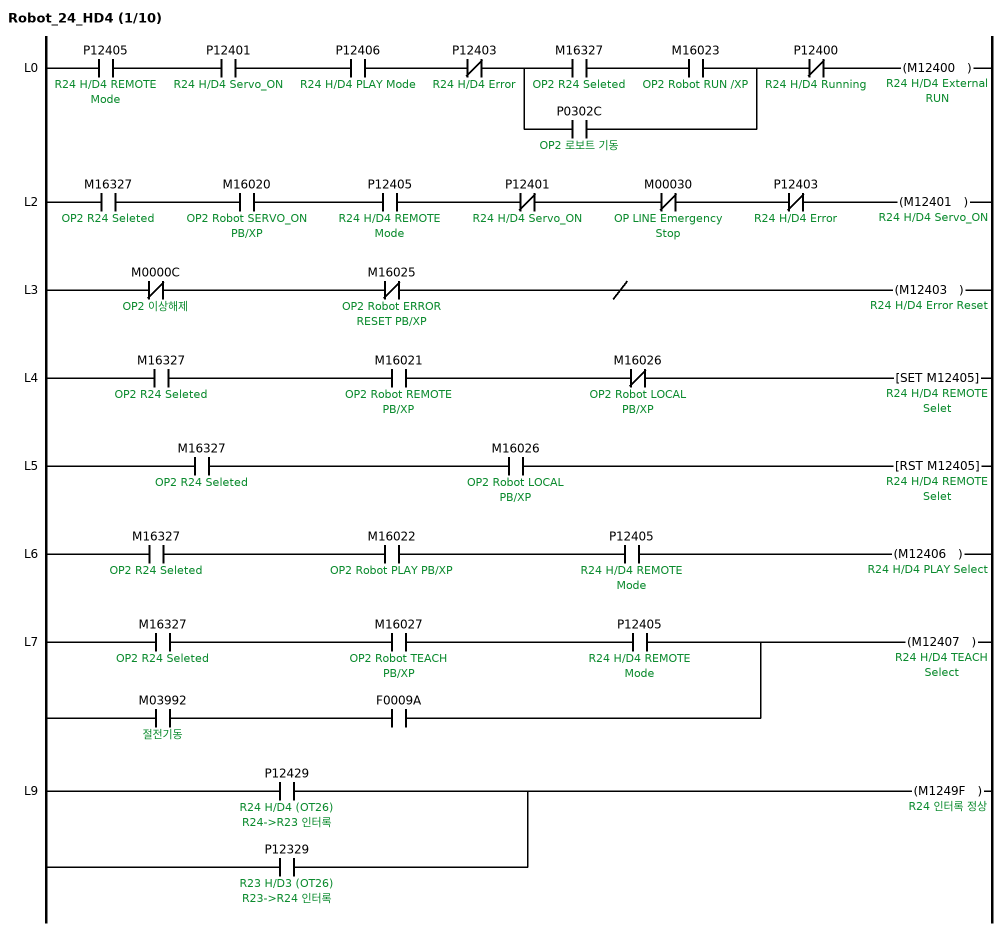
[picture p384: Robot_24_HD4 rungs L0-L9]
; L0
LOAD      P12405	// R24 H/D4 REMOTE Mode
AND       P12401	// R24 H/D4 Servo_ON
AND       P12406	// R24 H/D4 PLAY Mode
AND NOT   P12403	// R24 H/D4 Error
LOAD      M16327	// OP2 R24 Seleted
AND       M16023	// OP2 Robot RUN /XP
OR        P0302C	// OP2 로보트 기동
AND LOAD
AND NOT   P12400	// R24 H/D4 Running
OUT       M12400	// R24 H/D4 External RUN
; L2
LOAD      M16327	// OP2 R24 Seleted
AND       M16020	// OP2 Robot SERVO_ON PB/XP
AND       P12405	// R24 H/D4 REMOTE Mode
AND NOT   P12401	// R24 H/D4 Servo_ON
AND NOT   M00030	// OP LINE Emergency Stop
AND NOT   P12403	// R24 H/D4 Error
OUT       M12401	// R24 H/D4 Servo_ON
; L3
LOAD NOT  M0000C	// OP2 이상해제
AND NOT   M16025	// OP2 Robot ERROR RESET PB/XP
NOT
OUT       M12403	// R24 H/D4 Error Reset
; L4
LOAD      M16327	// OP2 R24 Seleted
AND       M16021	// OP2 Robot REMOTE PB/XP
AND NOT   M16026	// OP2 Robot LOCAL PB/XP
SET       M12405	// R24 H/D4 REMOTE Selet
; L5
LOAD      M16327	// OP2 R24 Seleted
AND       M16026	// OP2 Robot LOCAL PB/XP
RST       M12405	// R24 H/D4 REMOTE Selet
; L6
LOAD      M16327	// OP2 R24 Seleted
AND       M16022	// OP2 Robot PLAY PB/XP
AND       P12405	// R24 H/D4 REMOTE Mode
OUT       M12406	// R24 H/D4 PLAY Select
; L7
LOAD      M16327	// OP2 R24 Seleted
AND       M16027	// OP2 Robot TEACH PB/XP
AND       P12405	// R24 H/D4 REMOTE Mode
LOAD      M03992	// 절전기동
AND       F0009A
OR LOAD
OUT       M12407	// R24 H/D4 TEACH Select
; L9
LOAD      P12429	// R24 H/D4 (OT26) R24->R23 인터록
OR        P12329	// R23 H/D3 (OT26) R23->R24 인터록
OUT       M1249F	// R24 인터록 정상

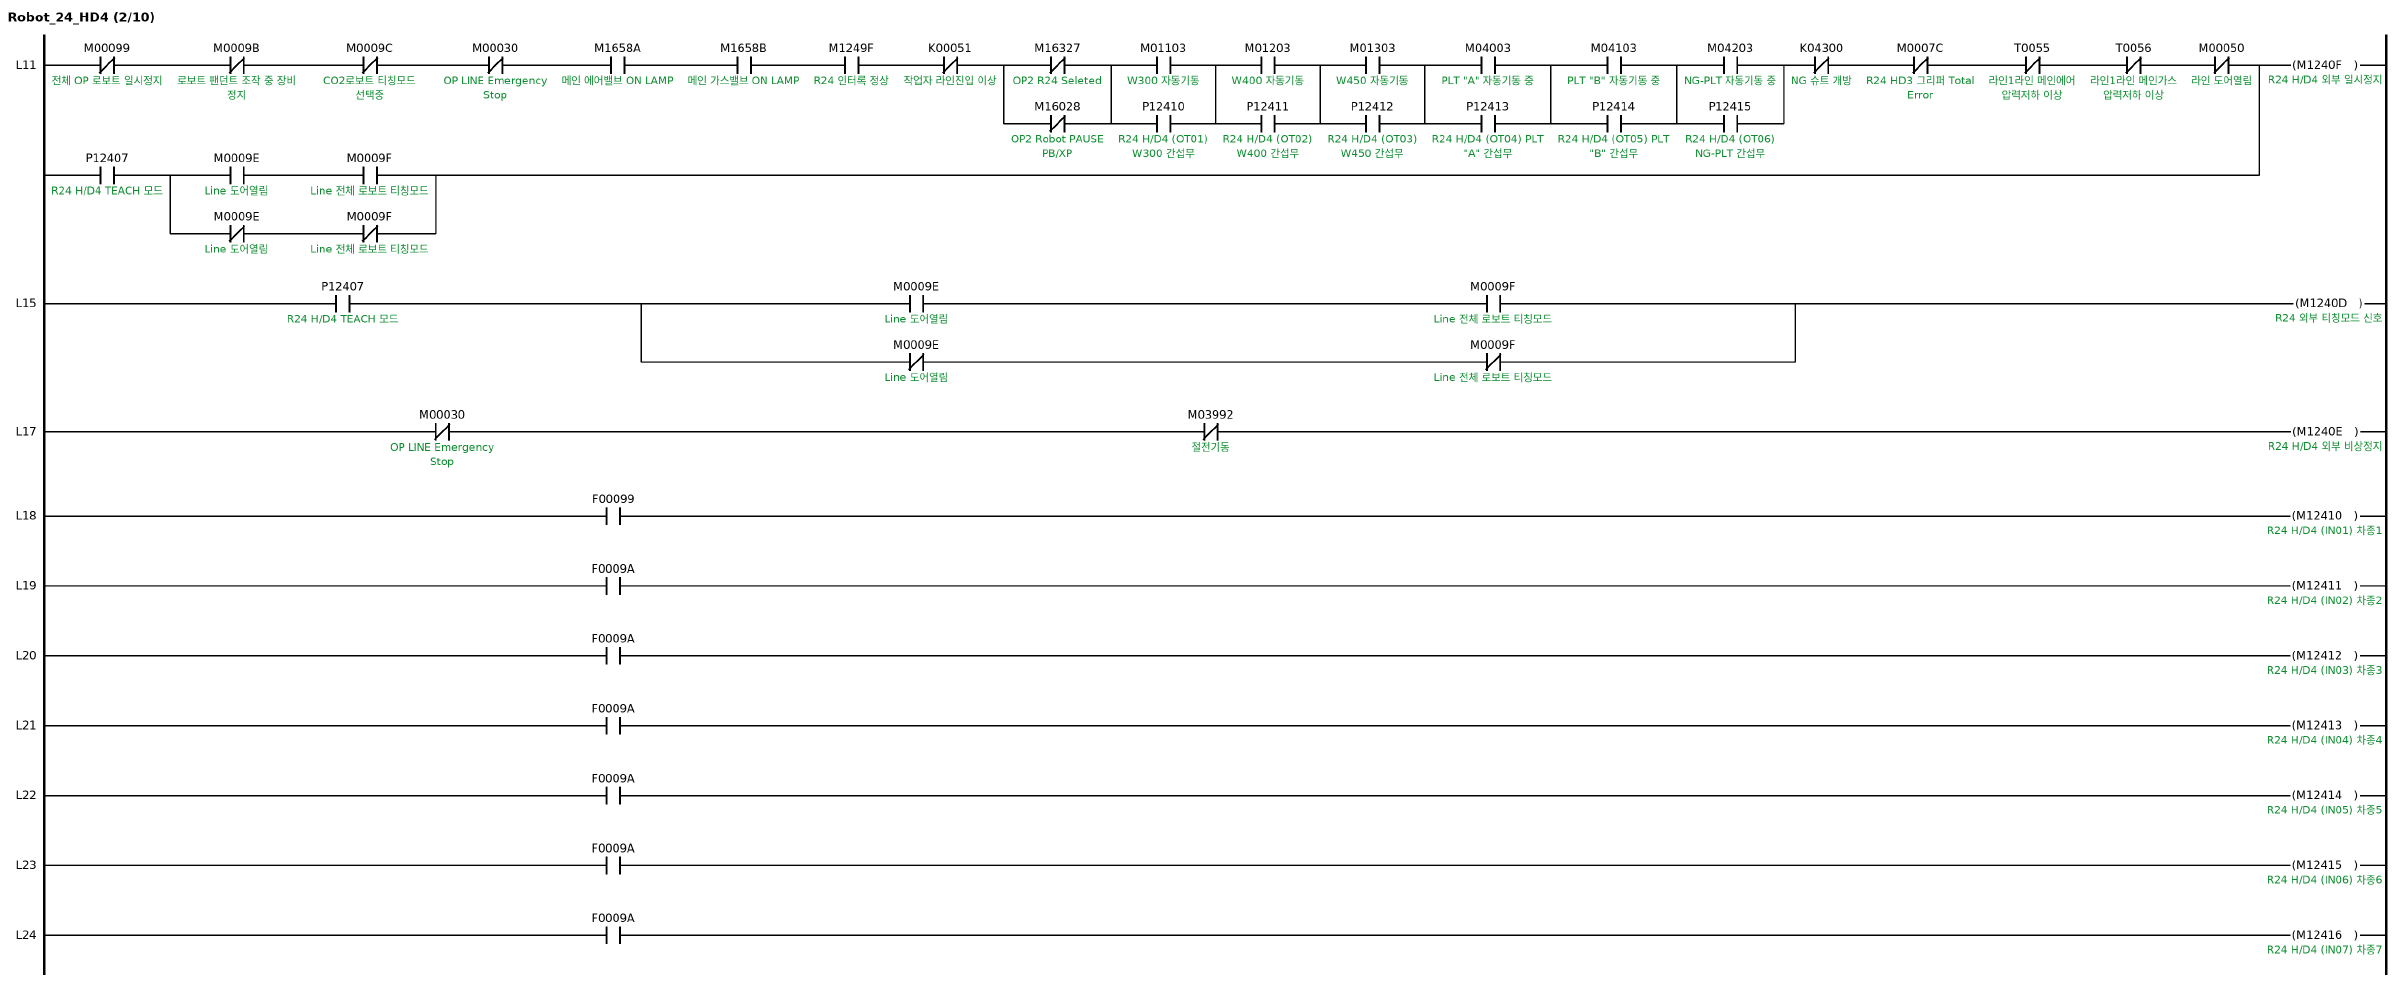
; L11
LOAD NOT  M00099	// 전체 OP 로보트 일시정지
AND NOT   M0009B	// 로보트 팬던트 조작 중 장비 정지
AND NOT   M0009C	// CO2로보트 티칭모드 선택중
AND NOT   M00030	// OP LINE Emergency Stop
AND       M1658A	// 메인 에어밸브 ON LAMP
AND       M1658B	// 메인 가스밸브 ON LAMP
AND       M1249F	// R24 인터록 정상
AND NOT   K00051	//  작업자 라인진입 이상
LOAD NOT  M16327	// OP2 R24 Seleted
OR NOT    M16028	// OP2 Robot PAUSE PB/XP
AND LOAD
LOAD      M01103	// W300 자동기동
OR        P12410	// R24 H/D4 (OT01) W300 간섭무
AND LOAD
LOAD      M01203	// W400 자동기동
OR        P12411	// R24 H/D4 (OT02) W400 간섭무
AND LOAD
LOAD      M01303	// W450 자동기동
OR        P12412	// R24 H/D4 (OT03) W450 간섭무
AND LOAD
LOAD      M04003	// PLT "A" 자동기동 중
OR        P12413	// R24 H/D4 (OT04) PLT "A" 간섭무
AND LOAD
LOAD      M04103	// PLT "B" 자동기동 중
OR        P12414	// R24 H/D4 (OT05) PLT "B" 간섭무
AND LOAD
LOAD      M04203	// NG-PLT 자동기동 중
OR        P12415	// R24 H/D4 (OT06) NG-PLT 간섭무
AND LOAD
AND NOT   K04300	// NG 슈트 개방
AND NOT   M0007C	// R24 HD3 그리퍼 Total Error 
AND NOT   T0055	// 라인1라인 메인에어 압력저하 이상
AND NOT   T0056	// 라인1라인 메인가스 압력저하 이상
AND NOT   M00050	// 라인 도어열림
LOAD      P12407	// R24 H/D4 TEACH 모드
LOAD      M0009E	// Line 도어열림
AND       M0009F	// Line 전체 로보트 티칭모드
LOAD NOT  M0009E	// Line 도어열림
AND NOT   M0009F	// Line 전체 로보트 티칭모드
OR LOAD
AND LOAD
OR LOAD
OUT       M1240F	// R24 H/D4 외부 일시정지
; L15
LOAD      P12407	// R24 H/D4 TEACH 모드
LOAD      M0009E	// Line 도어열림
AND       M0009F	// Line 전체 로보트 티칭모드
LOAD NOT  M0009E	// Line 도어열림
AND NOT   M0009F	// Line 전체 로보트 티칭모드
OR LOAD
AND LOAD
OUT       M1240D	// R24 외부 티칭모드 신호
; L17
LOAD NOT  M00030	// OP LINE Emergency Stop
AND NOT   M03992	// 절전기동
OUT       M1240E	// R24 H/D4 외부 비상정지 
; L18
LOAD      F00099
OUT       M12410	// R24 H/D4 (IN01) 차종1
; L19
LOAD      F0009A
OUT       M12411	// R24 H/D4 (IN02) 차종2
; L20
LOAD      F0009A
OUT       M12412	// R24 H/D4 (IN03) 차종3
; L21
LOAD      F0009A
OUT       M12413	// R24 H/D4 (IN04) 차종4
; L22
LOAD      F0009A
OUT       M12414	// R24 H/D4 (IN05) 차종5
; L23
LOAD      F0009A
OUT       M12415	// R24 H/D4 (IN06) 차종6
; L24
LOAD      F0009A
OUT       M12416	// R24 H/D4 (IN07) 차종7

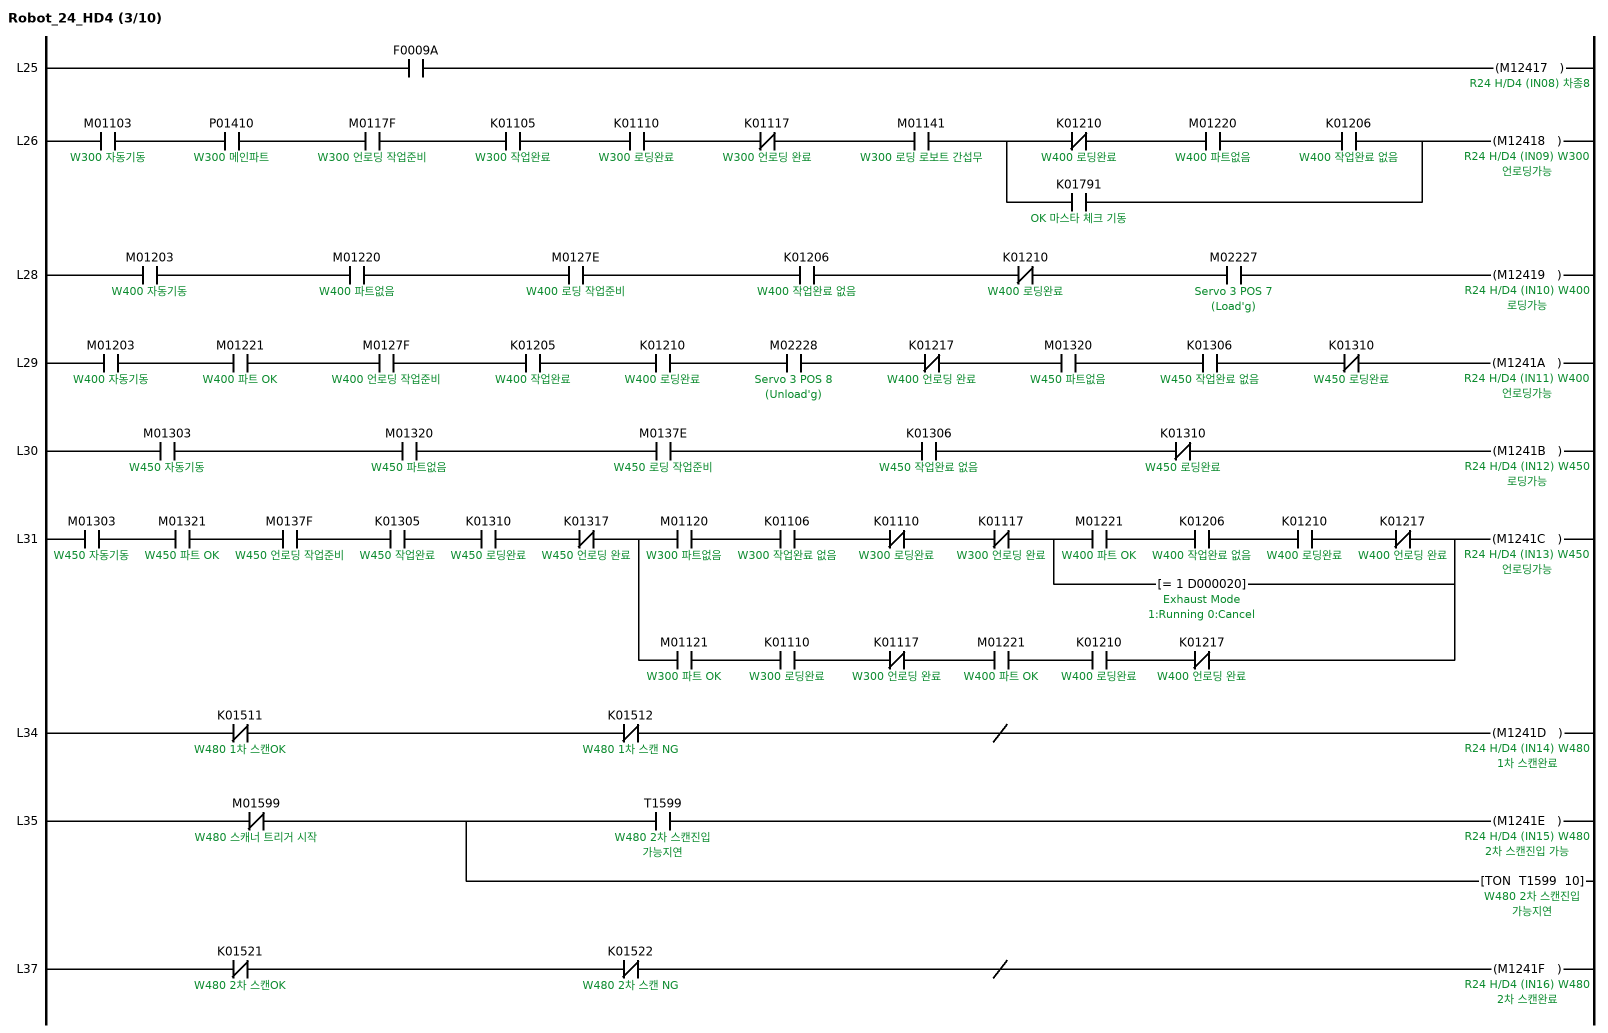
; L25
LOAD      F0009A
OUT       M12417	// R24 H/D4 (IN08) 차종8
; L26
LOAD      M01103	// W300 자동기동
AND       P01410	// W300 메인파트
AND       M0117F	// W300 언로딩 작업준비
AND       K01105	// W300 작업완료
AND       K01110	// W300 로딩완료
AND NOT   K01117	// W300 언로딩 완료
AND       M01141	// W300 로딩 로보트 간섭무
LOAD NOT  K01210	// W400 로딩완료
AND       M01220	// W400 파트없음
AND       K01206	// W400 작업완료 없음
OR        K01791	// OK 마스타 체크 기동
AND LOAD
OUT       M12418	// R24 H/D4 (IN09) W300 언로딩가능
; L28
LOAD      M01203	// W400 자동기동
AND       M01220	// W400 파트없음
AND       M0127E	// W400 로딩 작업준비
AND       K01206	// W400 작업완료 없음
AND NOT   K01210	// W400 로딩완료
AND       M02227	// Servo 3 POS 7 (Load'g)
OUT       M12419	// R24 H/D4 (IN10) W400 로딩가능
; L29
LOAD      M01203	// W400 자동기동
AND       M01221	// W400 파트 OK
AND       M0127F	// W400 언로딩 작업준비
AND       K01205	// W400 작업완료
AND       K01210	// W400 로딩완료
AND       M02228	// Servo 3 POS 8 (Unload'g)
AND NOT   K01217	// W400 언로딩 완료
AND       M01320	// W450 파트없음
AND       K01306	// W450 작업완료 없음
AND NOT   K01310	// W450 로딩완료
OUT       M1241A	// R24 H/D4 (IN11) W400 언로딩가능
; L30
LOAD      M01303	// W450 자동기동
AND       M01320	// W450 파트없음
AND       M0137E	// W450 로딩 작업준비
AND       K01306	// W450 작업완료 없음
AND NOT   K01310	// W450 로딩완료
OUT       M1241B	// R24 H/D4 (IN12) W450 로딩가능
; L31
LOAD      M01303	// W450 자동기동
AND       M01321	// W450 파트 OK
AND       M0137F	// W450 언로딩 작업준비
AND       K01305	// W450 작업완료
AND       K01310	// W450 로딩완료
AND NOT   K01317	// W450 언로딩 완료
LOAD      M01120	// W300 파트없음
AND       K01106	// W300 작업완료 없음
AND NOT   K01110	// W300 로딩완료
AND NOT   K01117	// W300 언로딩 완료
LOAD      M01221	// W400 파트 OK
AND       K01206	// W400 작업완료 없음
AND       K01210	// W400 로딩완료
AND NOT   K01217	// W400 언로딩 완료
OR=       1 D000020	// Exhaust Mode 1:Running 0:Cancel
AND LOAD
LOAD      M01121	// W300 파트 OK
AND       K01110	// W300 로딩완료
AND NOT   K01117	// W300 언로딩 완료
AND       M01221	// W400 파트 OK
AND       K01210	// W400 로딩완료
AND NOT   K01217	// W400 언로딩 완료
OR LOAD
AND LOAD
OUT       M1241C	// R24 H/D4 (IN13) W450 언로딩가능
; L34
LOAD NOT  K01511	// W480 1차 스캔OK
AND NOT   K01512	// W480 1차 스캔 NG
NOT
OUT       M1241D	// R24 H/D4 (IN14) W480 1차 스캔완료
; L35
LOAD NOT  M01599	// W480 스캐너 트리거 시작
MPUSH
AND       T1599	// W480 2차 스캔진입 가능지연
OUT       M1241E	// R24 H/D4 (IN15) W480 2차 스캔진입 가능
MPOP
TON       T1599 10	// W480 2차 스캔진입 가능지연
; L37
LOAD NOT  K01521	// W480 2차 스캔OK
AND NOT   K01522	// W480 2차 스캔 NG
NOT
OUT       M1241F	// R24 H/D4 (IN16) W480 2차 스캔완료

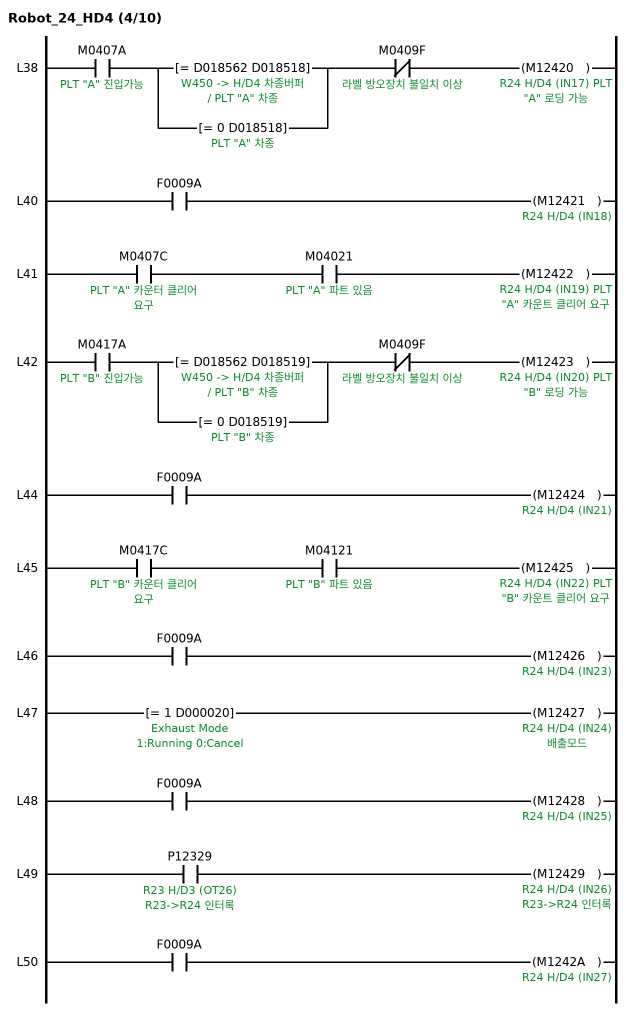
; L38
LOAD      M0407A	// PLT "A" 진입가능
LOAD=     D018562 D018518	// W450 -> H/D4 차종버퍼 / PLT "A" 차종
OR=       0 D018518	// PLT "A" 차종
AND LOAD
AND NOT   M0409F	// 라벨 방오장치 불일치 이상
OUT       M12420	// R24 H/D4 (IN17) PLT "A" 로딩 가능
; L40
LOAD      F0009A
OUT       M12421	// R24 H/D4 (IN18)
; L41
LOAD      M0407C	// PLT "A" 카운터 클리어 요구
AND       M04021	// PLT "A" 파트 있음
OUT       M12422	// R24 H/D4 (IN19) PLT "A" 카운트 클리어 요구
; L42
LOAD      M0417A	// PLT "B" 진입가능
LOAD=     D018562 D018519	// W450 -> H/D4 차종버퍼 / PLT "B" 차종
OR=       0 D018519	// PLT "B" 차종
AND LOAD
AND NOT   M0409F	// 라벨 방오장치 불일치 이상
OUT       M12423	// R24 H/D4 (IN20) PLT "B" 로딩 가능
; L44
LOAD      F0009A
OUT       M12424	// R24 H/D4 (IN21)
; L45
LOAD      M0417C	// PLT "B" 카운터 클리어 요구
AND       M04121	// PLT "B" 파트 있음
OUT       M12425	// R24 H/D4 (IN22) PLT "B" 카운트 클리어 요구
; L46
LOAD      F0009A
OUT       M12426	// R24 H/D4 (IN23)
; L47
LOAD=     1 D000020	// Exhaust Mode 1:Running 0:Cancel
OUT       M12427	// R24 H/D4 (IN24) 배출모드
; L48
LOAD      F0009A
OUT       M12428	// R24 H/D4 (IN25)
; L49
LOAD      P12329	// R23 H/D3 (OT26) R23->R24 인터록
OUT       M12429	// R24 H/D4 (IN26) R23->R24 인터록
; L50
LOAD      F0009A
OUT       M1242A	// R24 H/D4 (IN27)

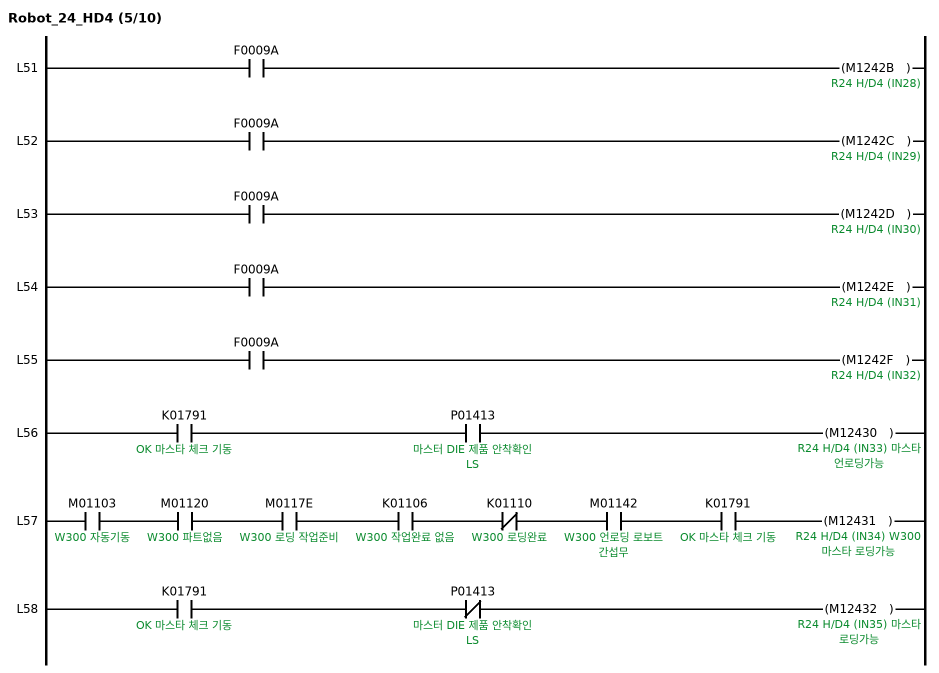
; L51
LOAD      F0009A
OUT       M1242B	// R24 H/D4 (IN28)
; L52
LOAD      F0009A
OUT       M1242C	// R24 H/D4 (IN29)
; L53
LOAD      F0009A
OUT       M1242D	// R24 H/D4 (IN30)
; L54
LOAD      F0009A
OUT       M1242E	// R24 H/D4 (IN31)
; L55
LOAD      F0009A
OUT       M1242F	// R24 H/D4 (IN32)
; L56
LOAD      K01791	// OK 마스타 체크 기동
AND       P01413	// 마스터 DIE 제품 안착확인 LS
OUT       M12430	// R24 H/D4 (IN33) 마스타 언로딩가능
; L57
LOAD      M01103	// W300 자동기동
AND       M01120	// W300 파트없음
AND       M0117E	// W300 로딩 작업준비
AND       K01106	// W300 작업완료 없음
AND NOT   K01110	// W300 로딩완료
AND       M01142	// W300 언로딩 로보트 간섭무
AND       K01791	// OK 마스타 체크 기동
OUT       M12431	// R24 H/D4 (IN34) W300 마스타 로딩가능
; L58
LOAD      K01791	// OK 마스타 체크 기동
AND NOT   P01413	// 마스터 DIE 제품 안착확인 LS
OUT       M12432	// R24 H/D4 (IN35) 마스타 로딩가능

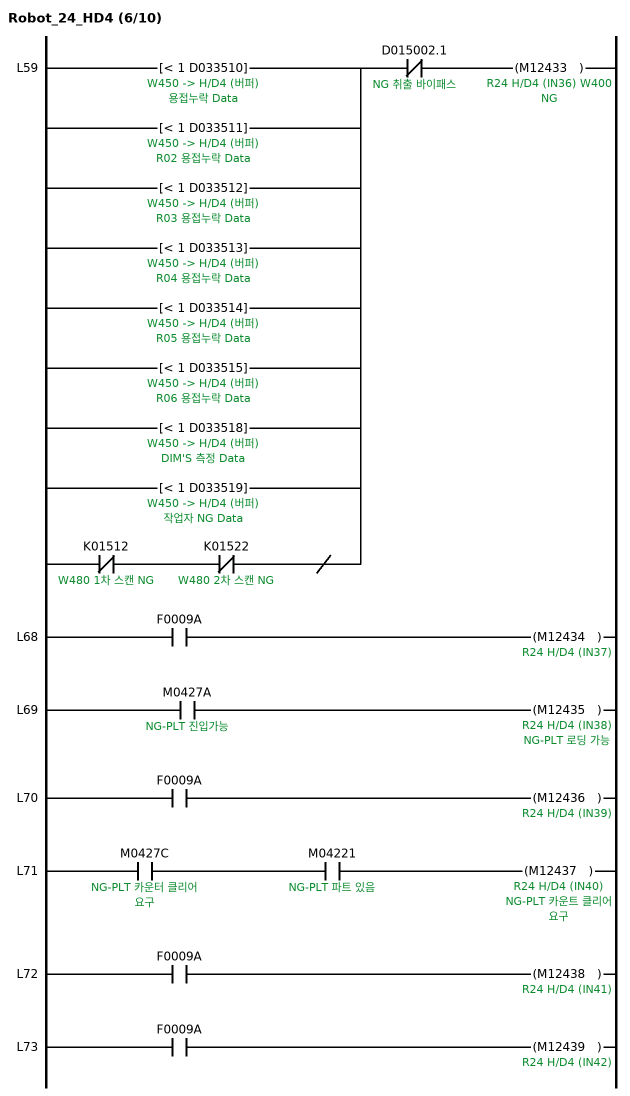
; L59
LOAD<     1 D033510	// W450 -> H/D4 (버퍼) 용접누락 Data
OR<       1 D033511	// W450 -> H/D4 (버퍼) R02 용접누락 Data
OR<       1 D033512	// W450 -> H/D4 (버퍼) R03 용접누락 Data
OR<       1 D033513	// W450 -> H/D4 (버퍼) R04 용접누락 Data
OR<       1 D033514	// W450 -> H/D4 (버퍼) R05 용접누락 Data
OR<       1 D033515	// W450 -> H/D4 (버퍼) R06 용접누락 Data
OR<       1 D033518	// W450 -> H/D4 (버퍼) DIM'S 측정 Data
OR<       1 D033519	// W450 -> H/D4 (버퍼) 작업자 NG Data
LOAD NOT  K01512	// W480 1차 스캔 NG
AND NOT   K01522	// W480 2차 스캔 NG
NOT
OR LOAD
AND NOT   D015002.1	// NG 취출 바이패스
OUT       M12433	// R24 H/D4 (IN36) W400 NG
; L68
LOAD      F0009A
OUT       M12434	// R24 H/D4 (IN37)
; L69
LOAD      M0427A	// NG-PLT 진입가능
OUT       M12435	// R24 H/D4 (IN38) NG-PLT 로딩 가능
; L70
LOAD      F0009A
OUT       M12436	// R24 H/D4 (IN39)
; L71
LOAD      M0427C	// NG-PLT 카운터 클리어 요구
AND       M04221	// NG-PLT 파트 있음
OUT       M12437	// R24 H/D4 (IN40) NG-PLT 카운트 클리어 요구
; L72
LOAD      F0009A
OUT       M12438	// R24 H/D4 (IN41)
; L73
LOAD      F0009A
OUT       M12439	// R24 H/D4 (IN42)

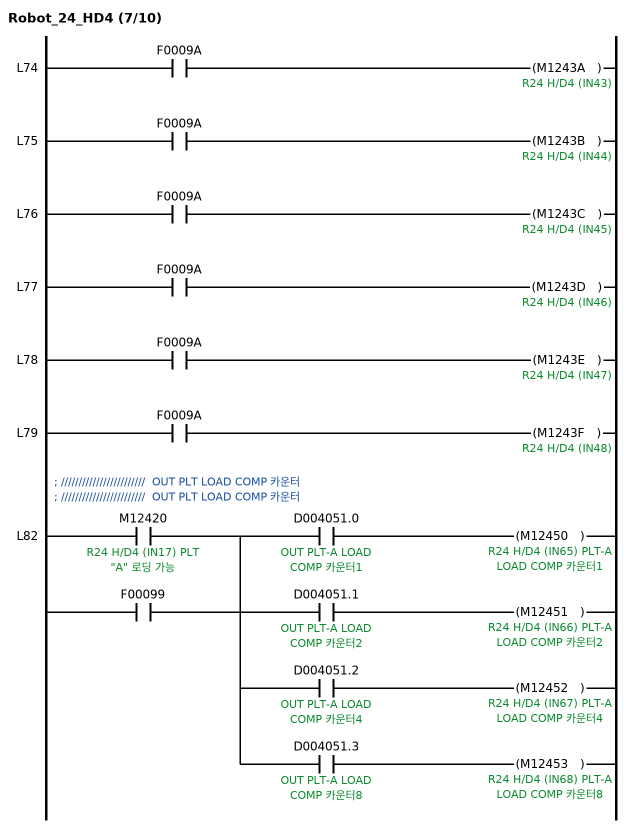
; L74
LOAD      F0009A
OUT       M1243A	// R24 H/D4 (IN43)
; L75
LOAD      F0009A
OUT       M1243B	// R24 H/D4 (IN44)
; L76
LOAD      F0009A
OUT       M1243C	// R24 H/D4 (IN45)
; L77
LOAD      F0009A
OUT       M1243D	// R24 H/D4 (IN46)
; L78
LOAD      F0009A
OUT       M1243E	// R24 H/D4 (IN47)
; L79
LOAD      F0009A
OUT       M1243F	// R24 H/D4 (IN48)
// ////////////////////////  OUT PLT LOAD COMP 카운터
// ////////////////////////  OUT PLT LOAD COMP 카운터
; L82
LOAD      M12420	// R24 H/D4 (IN17) PLT "A" 로딩 가능
OR        F00099
MPUSH
AND       D004051.0	// OUT PLT-A LOAD COMP 카운터1
OUT       M12450	// R24 H/D4 (IN65) PLT-A LOAD COMP 카운터1
MLOAD
AND       D004051.1	// OUT PLT-A LOAD COMP 카운터2
OUT       M12451	// R24 H/D4 (IN66) PLT-A LOAD COMP 카운터2
MLOAD
AND       D004051.2	// OUT PLT-A LOAD COMP 카운터4
OUT       M12452	// R24 H/D4 (IN67) PLT-A LOAD COMP 카운터4
MPOP
AND       D004051.3	// OUT PLT-A LOAD COMP 카운터8
OUT       M12453	// R24 H/D4 (IN68) PLT-A LOAD COMP 카운터8

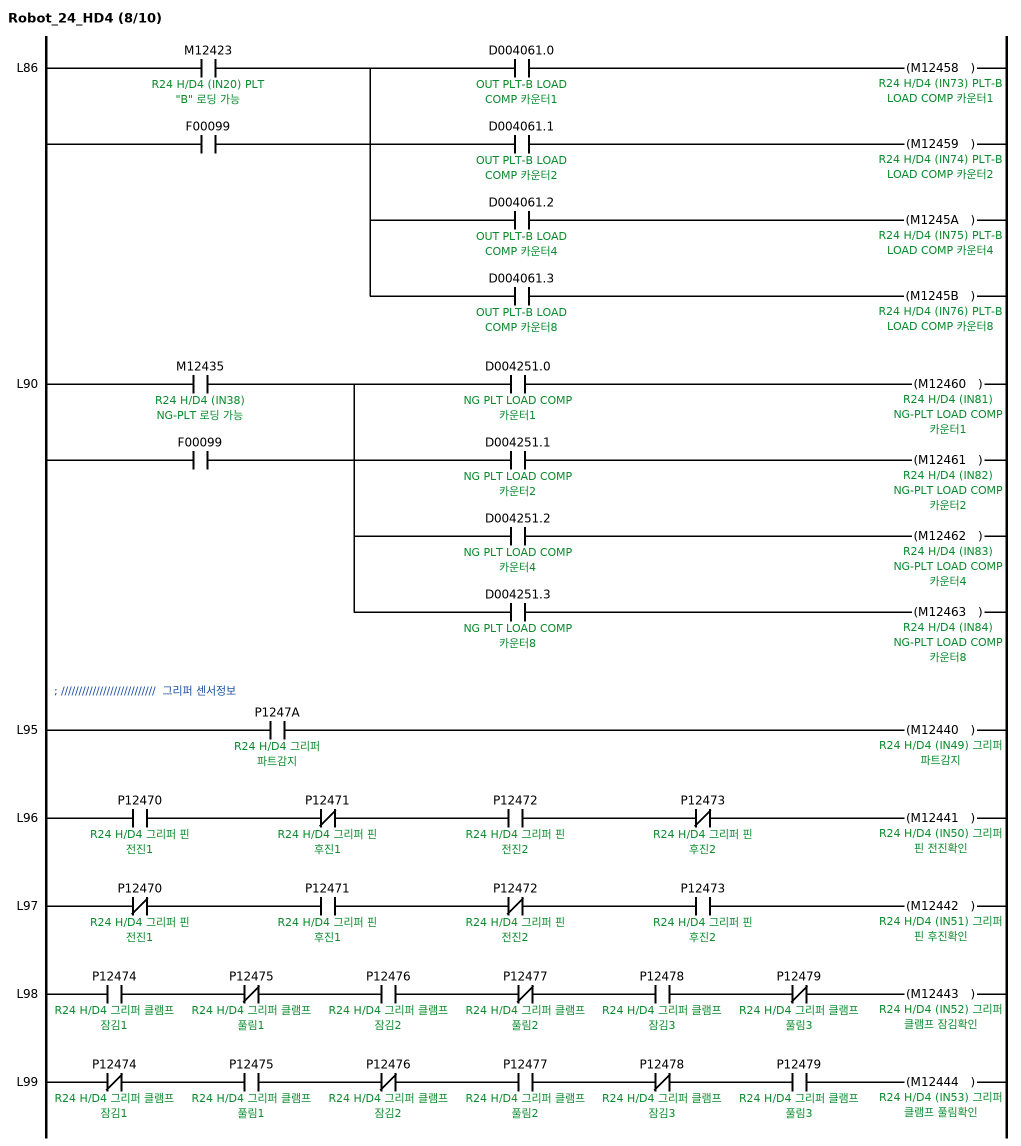
; L86
LOAD      M12423	// R24 H/D4 (IN20) PLT "B" 로딩 가능
OR        F00099
MPUSH
AND       D004061.0	// OUT PLT-B LOAD COMP 카운터1
OUT       M12458	// R24 H/D4 (IN73) PLT-B LOAD COMP 카운터1
MLOAD
AND       D004061.1	// OUT PLT-B LOAD COMP 카운터2
OUT       M12459	// R24 H/D4 (IN74) PLT-B LOAD COMP 카운터2
MLOAD
AND       D004061.2	// OUT PLT-B LOAD COMP 카운터4
OUT       M1245A	// R24 H/D4 (IN75) PLT-B LOAD COMP 카운터4
MPOP
AND       D004061.3	// OUT PLT-B LOAD COMP 카운터8
OUT       M1245B	// R24 H/D4 (IN76) PLT-B LOAD COMP 카운터8
; L90
LOAD      M12435	// R24 H/D4 (IN38) NG-PLT 로딩 가능
OR        F00099
MPUSH
AND       D004251.0	// NG PLT LOAD COMP 카운터1
OUT       M12460	// R24 H/D4 (IN81) NG-PLT LOAD COMP 카운터1
MLOAD
AND       D004251.1	// NG PLT LOAD COMP 카운터2
OUT       M12461	// R24 H/D4 (IN82) NG-PLT LOAD COMP 카운터2
MLOAD
AND       D004251.2	// NG PLT LOAD COMP 카운터4
OUT       M12462	// R24 H/D4 (IN83) NG-PLT LOAD COMP 카운터4
MPOP
AND       D004251.3	// NG PLT LOAD COMP 카운터8
OUT       M12463	// R24 H/D4 (IN84) NG-PLT LOAD COMP 카운터8
// ///////////////////////////  그리퍼 센서정보
; L95
LOAD      P1247A	// R24 H/D4 그리퍼 파트감지
OUT       M12440	// R24 H/D4 (IN49) 그리퍼 파트감지
; L96
LOAD      P12470	// R24 H/D4 그리퍼 핀 전진1
AND NOT   P12471	// R24 H/D4 그리퍼 핀 후진1
AND       P12472	// R24 H/D4 그리퍼 핀 전진2
AND NOT   P12473	// R24 H/D4 그리퍼 핀 후진2
OUT       M12441	// R24 H/D4 (IN50) 그리퍼 핀 전진확인
; L97
LOAD NOT  P12470	// R24 H/D4 그리퍼 핀 전진1
AND       P12471	// R24 H/D4 그리퍼 핀 후진1
AND NOT   P12472	// R24 H/D4 그리퍼 핀 전진2
AND       P12473	// R24 H/D4 그리퍼 핀 후진2
OUT       M12442	// R24 H/D4 (IN51) 그리퍼 핀 후진확인
; L98
LOAD      P12474	// R24 H/D4 그리퍼 클램프 잠김1
AND NOT   P12475	// R24 H/D4 그리퍼 클램프 풀림1
AND       P12476	// R24 H/D4 그리퍼 클램프 잠김2
AND NOT   P12477	// R24 H/D4 그리퍼 클램프 풀림2
AND       P12478	// R24 H/D4 그리퍼 클램프 잠김3
AND NOT   P12479	// R24 H/D4 그리퍼 클램프 풀림3
OUT       M12443	// R24 H/D4 (IN52) 그리퍼 클램프 잠김확인
; L99
LOAD NOT  P12474	// R24 H/D4 그리퍼 클램프 잠김1
AND       P12475	// R24 H/D4 그리퍼 클램프 풀림1
AND NOT   P12476	// R24 H/D4 그리퍼 클램프 잠김2
AND       P12477	// R24 H/D4 그리퍼 클램프 풀림2
AND NOT   P12478	// R24 H/D4 그리퍼 클램프 잠김3
AND       P12479	// R24 H/D4 그리퍼 클램프 풀림3
OUT       M12444	// R24 H/D4 (IN53) 그리퍼 클램프 풀림확인

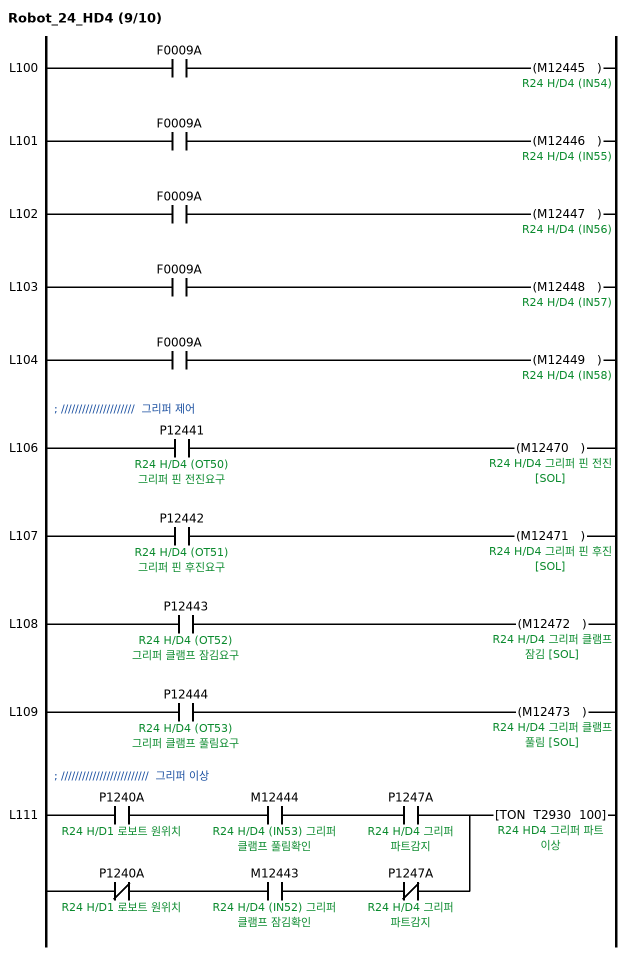
; L100
LOAD      F0009A
OUT       M12445	// R24 H/D4 (IN54)
; L101
LOAD      F0009A
OUT       M12446	// R24 H/D4 (IN55)
; L102
LOAD      F0009A
OUT       M12447	// R24 H/D4 (IN56)
; L103
LOAD      F0009A
OUT       M12448	// R24 H/D4 (IN57)
; L104
LOAD      F0009A
OUT       M12449	// R24 H/D4 (IN58)
// /////////////////////  그리퍼 제어
; L106
LOAD      P12441	// R24 H/D4 (OT50) 그리퍼 핀 전진요구
OUT       M12470	// R24 H/D4 그리퍼 핀 전진 [SOL]
; L107
LOAD      P12442	// R24 H/D4 (OT51) 그리퍼 핀 후진요구
OUT       M12471	// R24 H/D4 그리퍼 핀 후진 [SOL]
; L108
LOAD      P12443	// R24 H/D4 (OT52) 그리퍼 클램프 잠김요구
OUT       M12472	// R24 H/D4 그리퍼 클램프 잠김 [SOL]
; L109
LOAD      P12444	// R24 H/D4 (OT53) 그리퍼 클램프 풀림요구
OUT       M12473	// R24 H/D4 그리퍼 클램프 풀림 [SOL]
// /////////////////////////  그리퍼 이상
; L111
LOAD      P1240A	// R24 H/D1 로보트 원위치
AND       M12444	// R24 H/D4 (IN53) 그리퍼 클램프 풀림확인
AND       P1247A	// R24 H/D4 그리퍼 파트감지
LOAD NOT  P1240A	// R24 H/D1 로보트 원위치
AND       M12443	// R24 H/D4 (IN52) 그리퍼 클램프 잠김확인
AND NOT   P1247A	// R24 H/D4 그리퍼 파트감지
OR LOAD
TON       T2930 100	// R24 HD4 그리퍼 파트 이상

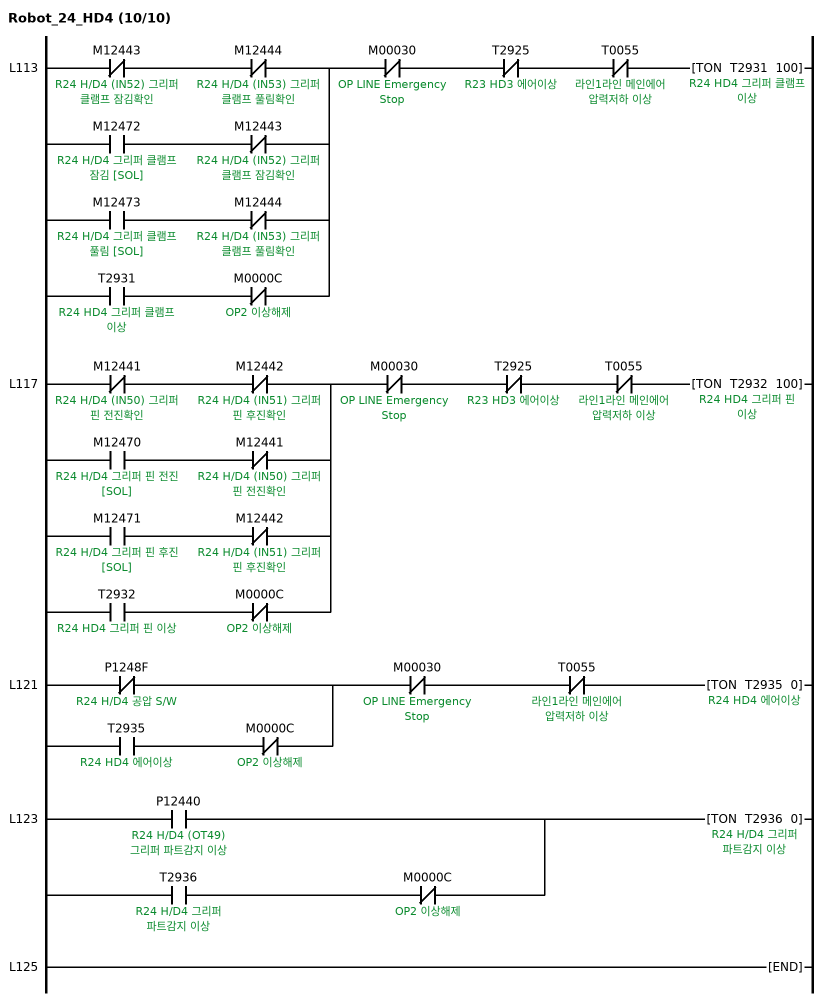
; L113
LOAD NOT  M12443	// R24 H/D4 (IN52) 그리퍼 클램프 잠김확인
AND NOT   M12444	// R24 H/D4 (IN53) 그리퍼 클램프 풀림확인
LOAD      M12472	// R24 H/D4 그리퍼 클램프 잠김 [SOL]
AND NOT   M12443	// R24 H/D4 (IN52) 그리퍼 클램프 잠김확인
OR LOAD
LOAD      M12473	// R24 H/D4 그리퍼 클램프 풀림 [SOL]
AND NOT   M12444	// R24 H/D4 (IN53) 그리퍼 클램프 풀림확인
OR LOAD
LOAD      T2931	// R24 HD4 그리퍼 클램프 이상
AND NOT   M0000C	// OP2 이상해제
OR LOAD
AND NOT   M00030	// OP LINE Emergency Stop
AND NOT   T2925	// R23 HD3 에어이상
AND NOT   T0055	// 라인1라인 메인에어 압력저하 이상
TON       T2931 100	// R24 HD4 그리퍼 클램프 이상
; L117
LOAD NOT  M12441	// R24 H/D4 (IN50) 그리퍼 핀 전진확인
AND NOT   M12442	// R24 H/D4 (IN51) 그리퍼 핀 후진확인
LOAD      M12470	// R24 H/D4 그리퍼 핀 전진 [SOL]
AND NOT   M12441	// R24 H/D4 (IN50) 그리퍼 핀 전진확인
OR LOAD
LOAD      M12471	// R24 H/D4 그리퍼 핀 후진 [SOL]
AND NOT   M12442	// R24 H/D4 (IN51) 그리퍼 핀 후진확인
OR LOAD
LOAD      T2932	// R24 HD4 그리퍼 핀 이상
AND NOT   M0000C	// OP2 이상해제
OR LOAD
AND NOT   M00030	// OP LINE Emergency Stop
AND NOT   T2925	// R23 HD3 에어이상
AND NOT   T0055	// 라인1라인 메인에어 압력저하 이상
TON       T2932 100	// R24 HD4 그리퍼 핀 이상
; L121
LOAD NOT  P1248F	// R24 H/D4 공압 S/W
LOAD      T2935	// R24 HD4 에어이상
AND NOT   M0000C	// OP2 이상해제
OR LOAD
AND NOT   M00030	// OP LINE Emergency Stop
AND NOT   T0055	// 라인1라인 메인에어 압력저하 이상
TON       T2935 0	// R24 HD4 에어이상
; L123
LOAD      P12440	// R24 H/D4 (OT49) 그리퍼 파트감지 이상
LOAD      T2936	// R24 H/D4 그리퍼 파트감지 이상
AND NOT   M0000C	// OP2 이상해제
OR LOAD
TON       T2936 0	// R24 H/D4 그리퍼 파트감지 이상
; L125
END

PROGRAM ARC관리 (task: 스캔 프로그램)

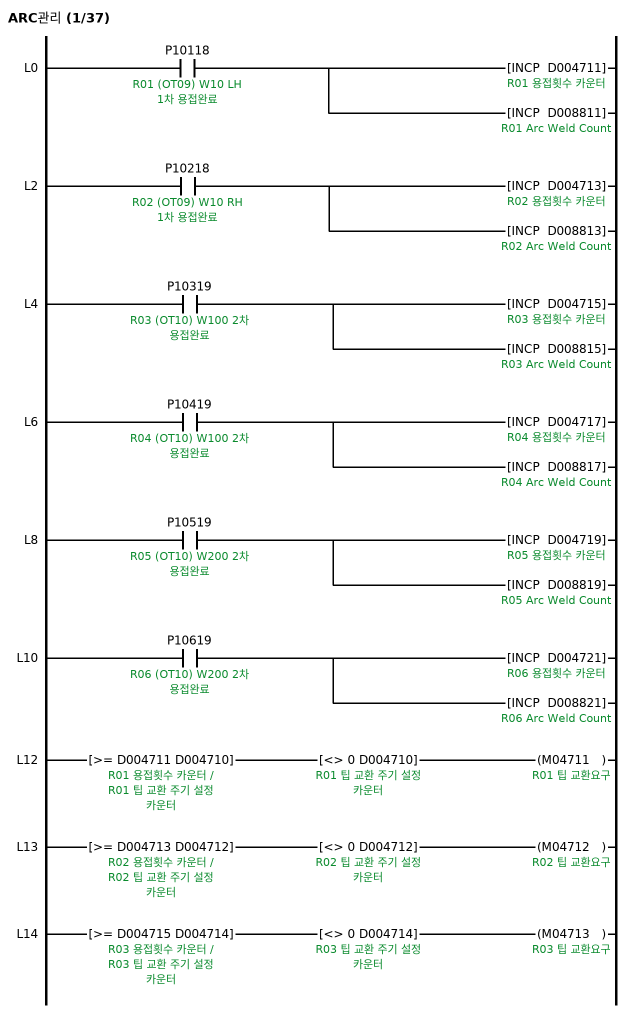
; L0
LOAD      P10118	// R01 (OT09) W10 LH 1차 용접완료
INCP      D004711	// R01 용접횟수 카운터
INCP      D008811	// R01 Arc Weld Count
; L2
LOAD      P10218	// R02 (OT09) W10 RH 1차 용접완료
INCP      D004713	// R02 용접횟수 카운터
INCP      D008813	// R02 Arc Weld Count
; L4
LOAD      P10319	// R03 (OT10) W100 2차 용접완료
INCP      D004715	// R03 용접횟수 카운터
INCP      D008815	// R03 Arc Weld Count
; L6
LOAD      P10419	// R04 (OT10) W100 2차 용접완료
INCP      D004717	// R04 용접횟수 카운터
INCP      D008817	// R04 Arc Weld Count
; L8
LOAD      P10519	// R05 (OT10) W200 2차 용접완료
INCP      D004719	// R05 용접횟수 카운터
INCP      D008819	// R05 Arc Weld Count
; L10
LOAD      P10619	// R06 (OT10) W200 2차 용접완료
INCP      D004721	// R06 용접횟수 카운터
INCP      D008821	// R06 Arc Weld Count
; L12
LOAD>=    D004711 D004710	// R01 용접횟수 카운터 / R01 팁 교환 주기 설정 카운터
AND<>     0 D004710	// R01 팁 교환 주기 설정 카운터
OUT       M04711	// R01 팁 교환요구
; L13
LOAD>=    D004713 D004712	// R02 용접횟수 카운터 / R02 팁 교환 주기 설정 카운터
AND<>     0 D004712	// R02 팁 교환 주기 설정 카운터
OUT       M04712	// R02 팁 교환요구
; L14
LOAD>=    D004715 D004714	// R03 용접횟수 카운터 / R03 팁 교환 주기 설정 카운터
AND<>     0 D004714	// R03 팁 교환 주기 설정 카운터
OUT       M04713	// R03 팁 교환요구

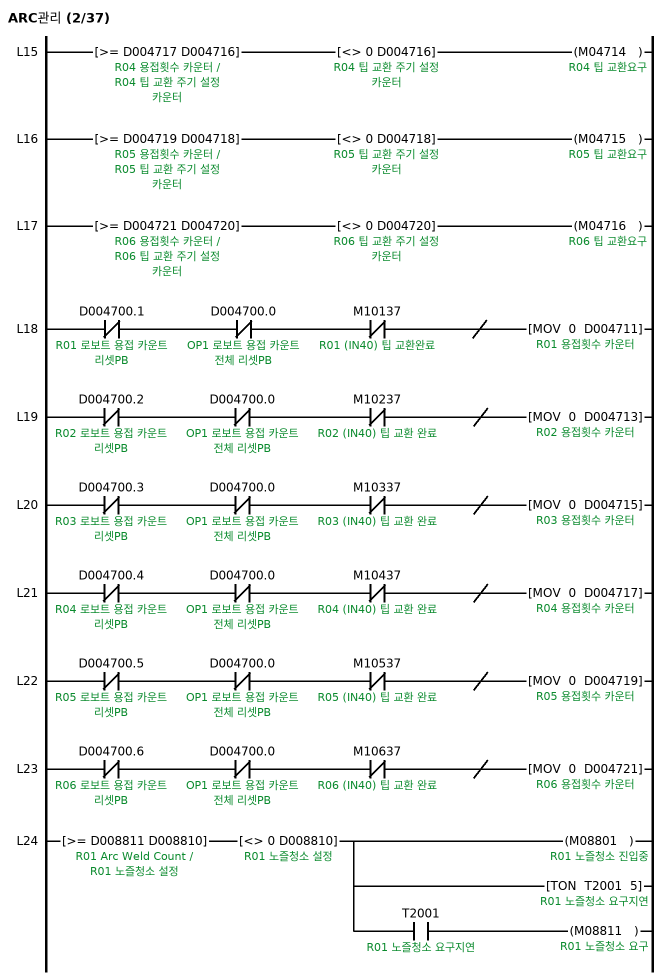
; L15
LOAD>=    D004717 D004716	// R04 용접횟수 카운터 / R04 팁 교환 주기 설정 카운터
AND<>     0 D004716	// R04 팁 교환 주기 설정 카운터
OUT       M04714	// R04 팁 교환요구
; L16
LOAD>=    D004719 D004718	// R05 용접횟수 카운터 / R05 팁 교환 주기 설정 카운터
AND<>     0 D004718	// R05 팁 교환 주기 설정 카운터
OUT       M04715	// R05 팁 교환요구
; L17
LOAD>=    D004721 D004720	// R06 용접횟수 카운터 / R06 팁 교환 주기 설정 카운터
AND<>     0 D004720	// R06 팁 교환 주기 설정 카운터
OUT       M04716	// R06 팁 교환요구
; L18
LOAD NOT  D004700.1	// R01 로보트 용접 카운트 리셋PB
AND NOT   D004700.0	// OP1 로보트 용접 카운트 전체 리셋PB
AND NOT   M10137	// R01 (IN40) 팁 교환완료
NOT
MOV       0 D004711	// R01 용접횟수 카운터
; L19
LOAD NOT  D004700.2	// R02 로보트 용접 카운트 리셋PB
AND NOT   D004700.0	// OP1 로보트 용접 카운트 전체 리셋PB
AND NOT   M10237	// R02 (IN40) 팁 교환 완료
NOT
MOV       0 D004713	// R02 용접횟수 카운터
; L20
LOAD NOT  D004700.3	// R03 로보트 용접 카운트 리셋PB
AND NOT   D004700.0	// OP1 로보트 용접 카운트 전체 리셋PB
AND NOT   M10337	// R03 (IN40) 팁 교환 완료
NOT
MOV       0 D004715	// R03 용접횟수 카운터
; L21
LOAD NOT  D004700.4	// R04 로보트 용접 카운트 리셋PB
AND NOT   D004700.0	// OP1 로보트 용접 카운트 전체 리셋PB
AND NOT   M10437	// R04 (IN40) 팁 교환 완료
NOT
MOV       0 D004717	// R04 용접횟수 카운터
; L22
LOAD NOT  D004700.5	// R05 로보트 용접 카운트 리셋PB
AND NOT   D004700.0	// OP1 로보트 용접 카운트 전체 리셋PB
AND NOT   M10537	// R05 (IN40) 팁 교환 완료
NOT
MOV       0 D004719	// R05 용접횟수 카운터
; L23
LOAD NOT  D004700.6	// R06 로보트 용접 카운트 리셋PB
AND NOT   D004700.0	// OP1 로보트 용접 카운트 전체 리셋PB
AND NOT   M10637	// R06 (IN40) 팁 교환 완료
NOT
MOV       0 D004721	// R06 용접횟수 카운터
; L24
LOAD>=    D008811 D008810	// R01 Arc Weld Count / R01 노즐청소 설정
AND<>     0 D008810	// R01 노즐청소 설정
OUT       M08801	// R01 노즐청소 진입중
TON       T2001 5	// R01 노즐청소 요구지연
AND       T2001	// R01 노즐청소 요구지연
OUT       M08811	// R01 노즐청소 요구

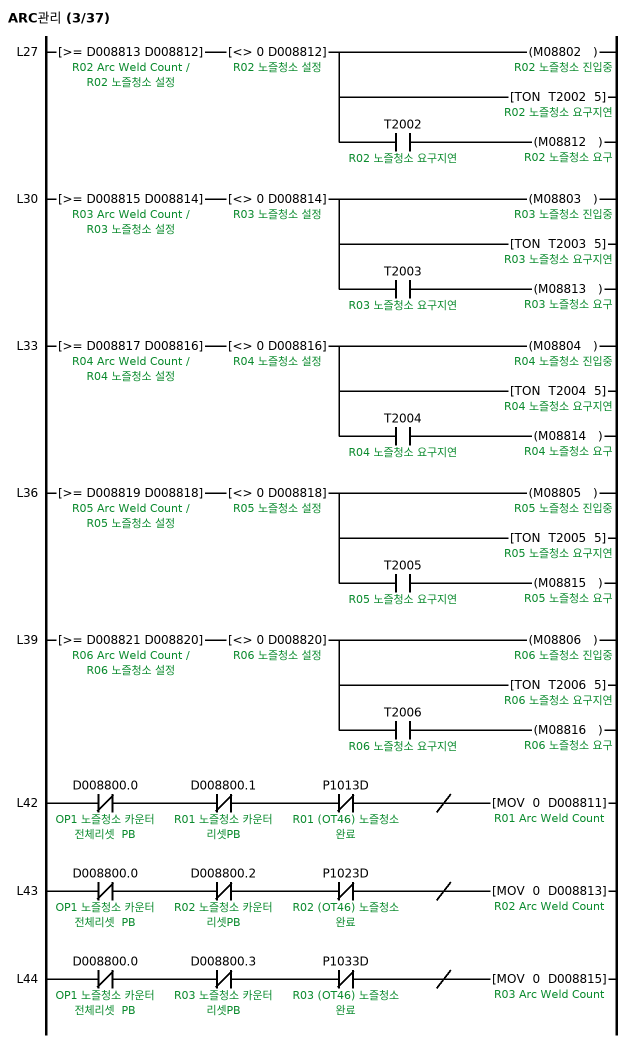
; L27
LOAD>=    D008813 D008812	// R02 Arc Weld Count / R02 노즐청소 설정
AND<>     0 D008812	// R02 노즐청소 설정
OUT       M08802	// R02 노즐청소 진입중
TON       T2002 5	// R02 노즐청소 요구지연
AND       T2002	// R02 노즐청소 요구지연
OUT       M08812	// R02 노즐청소 요구
; L30
LOAD>=    D008815 D008814	// R03 Arc Weld Count / R03 노즐청소 설정
AND<>     0 D008814	// R03 노즐청소 설정
OUT       M08803	// R03 노즐청소 진입중
TON       T2003 5	// R03 노즐청소 요구지연
AND       T2003	// R03 노즐청소 요구지연
OUT       M08813	// R03 노즐청소 요구
; L33
LOAD>=    D008817 D008816	// R04 Arc Weld Count / R04 노즐청소 설정
AND<>     0 D008816	// R04 노즐청소 설정
OUT       M08804	// R04 노즐청소 진입중
TON       T2004 5	// R04 노즐청소 요구지연
AND       T2004	// R04 노즐청소 요구지연
OUT       M08814	// R04 노즐청소 요구
; L36
LOAD>=    D008819 D008818	// R05 Arc Weld Count / R05 노즐청소 설정
AND<>     0 D008818	// R05 노즐청소 설정
OUT       M08805	// R05 노즐청소 진입중
TON       T2005 5	// R05 노즐청소 요구지연
AND       T2005	// R05 노즐청소 요구지연
OUT       M08815	// R05 노즐청소 요구
; L39
LOAD>=    D008821 D008820	// R06 Arc Weld Count / R06 노즐청소 설정
AND<>     0 D008820	// R06 노즐청소 설정
OUT       M08806	// R06 노즐청소 진입중
TON       T2006 5	// R06 노즐청소 요구지연
AND       T2006	// R06 노즐청소 요구지연
OUT       M08816	// R06 노즐청소 요구
; L42
LOAD NOT  D008800.0	// OP1 노즐청소 카운터 전체리셋  PB
AND NOT   D008800.1	// R01 노즐청소 카운터 리셋PB
AND NOT   P1013D	// R01 (OT46) 노즐청소 완료
NOT
MOV       0 D008811	// R01 Arc Weld Count
; L43
LOAD NOT  D008800.0	// OP1 노즐청소 카운터 전체리셋  PB
AND NOT   D008800.2	// R02 노즐청소 카운터 리셋PB
AND NOT   P1023D	// R02 (OT46) 노즐청소 완료
NOT
MOV       0 D008813	// R02 Arc Weld Count
; L44
LOAD NOT  D008800.0	// OP1 노즐청소 카운터 전체리셋  PB
AND NOT   D008800.3	// R03 노즐청소 카운터 리셋PB
AND NOT   P1033D	// R03 (OT46) 노즐청소 완료
NOT
MOV       0 D008815	// R03 Arc Weld Count

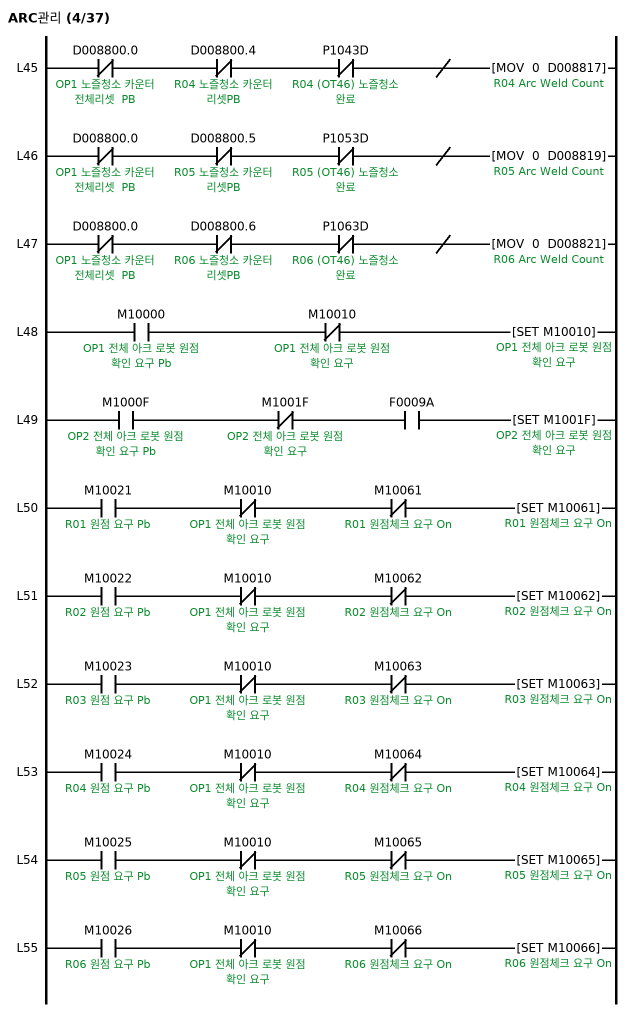
; L45
LOAD NOT  D008800.0	// OP1 노즐청소 카운터 전체리셋  PB
AND NOT   D008800.4	// R04 노즐청소 카운터 리셋PB
AND NOT   P1043D	// R04 (OT46) 노즐청소 완료
NOT
MOV       0 D008817	// R04 Arc Weld Count
; L46
LOAD NOT  D008800.0	// OP1 노즐청소 카운터 전체리셋  PB
AND NOT   D008800.5	// R05 노즐청소 카운터 리셋PB
AND NOT   P1053D	// R05 (OT46) 노즐청소 완료
NOT
MOV       0 D008819	// R05 Arc Weld Count
; L47
LOAD NOT  D008800.0	// OP1 노즐청소 카운터 전체리셋  PB
AND NOT   D008800.6	// R06 노즐청소 카운터 리셋PB
AND NOT   P1063D	// R06 (OT46) 노즐청소 완료
NOT
MOV       0 D008821	// R06 Arc Weld Count
; L48
LOAD      M10000	// OP1 전체 아크 로봇 원점 확인 요구 Pb
AND NOT   M10010	// OP1 전체 아크 로봇 원점 확인 요구
SET       M10010	// OP1 전체 아크 로봇 원점 확인 요구
; L49
LOAD      M1000F	// OP2 전체 아크 로봇 원점 확인 요구 Pb
AND NOT   M1001F	// OP2 전체 아크 로봇 원점 확인 요구
AND       F0009A
SET       M1001F	// OP2 전체 아크 로봇 원점 확인 요구
; L50
LOAD      M10021	// R01 원점 요구 Pb
AND NOT   M10010	// OP1 전체 아크 로봇 원점 확인 요구
AND NOT   M10061	// R01 원점체크 요구 On
SET       M10061	// R01 원점체크 요구 On
; L51
LOAD      M10022	// R02 원점 요구 Pb
AND NOT   M10010	// OP1 전체 아크 로봇 원점 확인 요구
AND NOT   M10062	// R02 원점체크 요구 On
SET       M10062	// R02 원점체크 요구 On
; L52
LOAD      M10023	// R03 원점 요구 Pb
AND NOT   M10010	// OP1 전체 아크 로봇 원점 확인 요구
AND NOT   M10063	// R03 원점체크 요구 On
SET       M10063	// R03 원점체크 요구 On
; L53
LOAD      M10024	// R04 원점 요구 Pb
AND NOT   M10010	// OP1 전체 아크 로봇 원점 확인 요구
AND NOT   M10064	// R04 원점체크 요구 On
SET       M10064	// R04 원점체크 요구 On
; L54
LOAD      M10025	// R05 원점 요구 Pb
AND NOT   M10010	// OP1 전체 아크 로봇 원점 확인 요구
AND NOT   M10065	// R05 원점체크 요구 On
SET       M10065	// R05 원점체크 요구 On
; L55
LOAD      M10026	// R06 원점 요구 Pb
AND NOT   M10010	// OP1 전체 아크 로봇 원점 확인 요구
AND NOT   M10066	// R06 원점체크 요구 On
SET       M10066	// R06 원점체크 요구 On

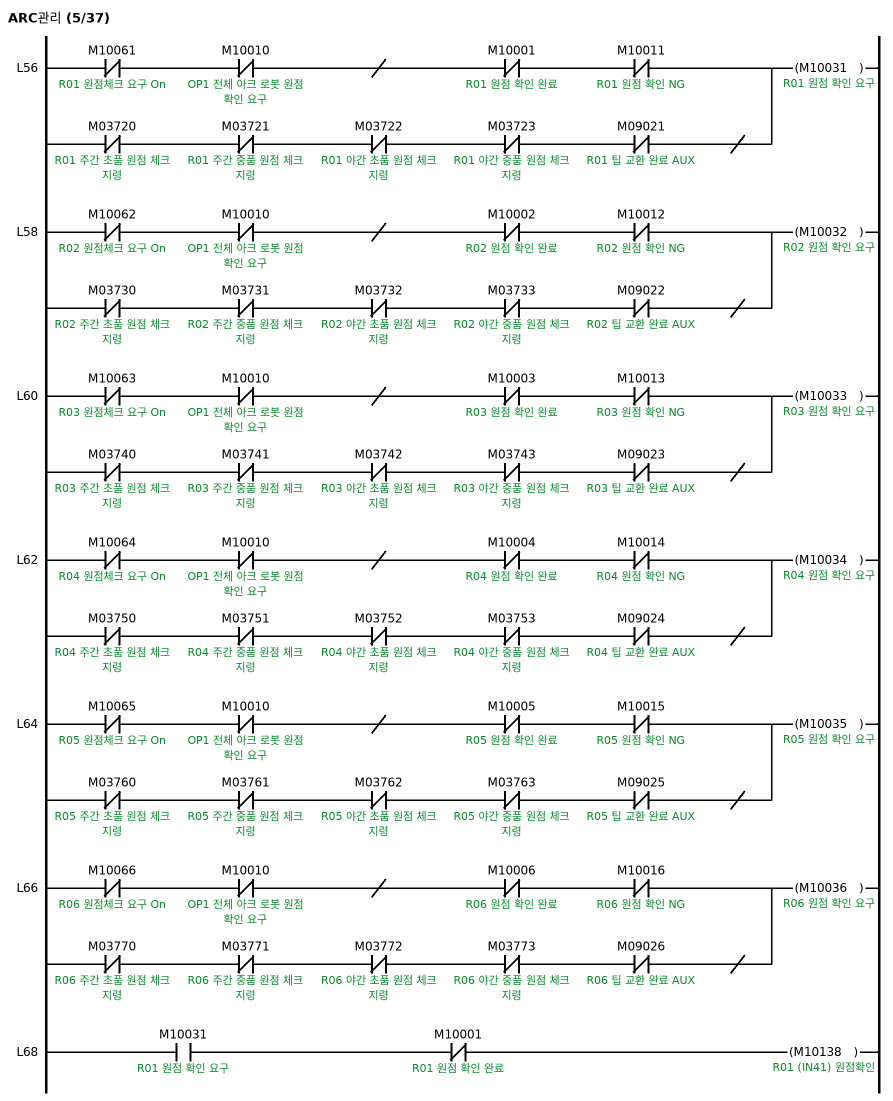
; L56
LOAD NOT  M10061	// R01 원점체크 요구 On
AND NOT   M10010	// OP1 전체 아크 로봇 원점 확인 요구
NOT
AND NOT   M10001	// R01 원점 확인 완료
AND NOT   M10011	// R01 원점 확인 NG
LOAD NOT  M03720	// R01 주간 초품 원점 체크 지령
AND NOT   M03721	// R01 주간 중품 원점 체크 지령
AND NOT   M03722	// R01 야간 초품 원점 체크 지령
AND NOT   M03723	// R01 야간 중품 원점 체크 지령
AND NOT   M09021	// R01 팁 교환 완료 AUX
NOT
OR LOAD
OUT       M10031	// R01 원점 확인 요구
; L58
LOAD NOT  M10062	// R02 원점체크 요구 On
AND NOT   M10010	// OP1 전체 아크 로봇 원점 확인 요구
NOT
AND NOT   M10002	// R02 원점 확인 완료
AND NOT   M10012	// R02 원점 확인 NG
LOAD NOT  M03730	// R02 주간 초품 원점 체크 지령
AND NOT   M03731	// R02 주간 중품 원점 체크 지령
AND NOT   M03732	// R02 야간 초품 원점 체크 지령
AND NOT   M03733	// R02 야간 중품 원점 체크 지령
AND NOT   M09022	// R02 팁 교환 완료 AUX
NOT
OR LOAD
OUT       M10032	// R02 원점 확인 요구
; L60
LOAD NOT  M10063	// R03 원점체크 요구 On
AND NOT   M10010	// OP1 전체 아크 로봇 원점 확인 요구
NOT
AND NOT   M10003	// R03 원점 확인 완료
AND NOT   M10013	// R03 원점 확인 NG
LOAD NOT  M03740	// R03 주간 초품 원점 체크 지령
AND NOT   M03741	// R03 주간 중품 원점 체크 지령
AND NOT   M03742	// R03 야간 초품 원점 체크 지령
AND NOT   M03743	// R03 야간 중품 원점 체크 지령
AND NOT   M09023	// R03 팁 교환 완료 AUX
NOT
OR LOAD
OUT       M10033	// R03 원점 확인 요구
; L62
LOAD NOT  M10064	// R04 원점체크 요구 On
AND NOT   M10010	// OP1 전체 아크 로봇 원점 확인 요구
NOT
AND NOT   M10004	// R04 원점 확인 완료
AND NOT   M10014	// R04 원점 확인 NG
LOAD NOT  M03750	// R04 주간 초품 원점 체크 지령
AND NOT   M03751	// R04 주간 중품 원점 체크 지령
AND NOT   M03752	// R04 야간 초품 원점 체크 지령
AND NOT   M03753	// R04 야간 중품 원점 체크 지령
AND NOT   M09024	// R04 팁 교환 완료 AUX
NOT
OR LOAD
OUT       M10034	// R04 원점 확인 요구
; L64
LOAD NOT  M10065	// R05 원점체크 요구 On
AND NOT   M10010	// OP1 전체 아크 로봇 원점 확인 요구
NOT
AND NOT   M10005	// R05 원점 확인 완료
AND NOT   M10015	// R05 원점 확인 NG
LOAD NOT  M03760	// R05 주간 초품 원점 체크 지령
AND NOT   M03761	// R05 주간 중품 원점 체크 지령
AND NOT   M03762	// R05 야간 초품 원점 체크 지령
AND NOT   M03763	// R05 야간 중품 원점 체크 지령
AND NOT   M09025	// R05 팁 교환 완료 AUX
NOT
OR LOAD
OUT       M10035	// R05 원점 확인 요구
; L66
LOAD NOT  M10066	// R06 원점체크 요구 On
AND NOT   M10010	// OP1 전체 아크 로봇 원점 확인 요구
NOT
AND NOT   M10006	// R06 원점 확인 완료
AND NOT   M10016	// R06 원점 확인 NG
LOAD NOT  M03770	// R06 주간 초품 원점 체크 지령
AND NOT   M03771	// R06 주간 중품 원점 체크 지령
AND NOT   M03772	// R06 야간 초품 원점 체크 지령
AND NOT   M03773	// R06 야간 중품 원점 체크 지령
AND NOT   M09026	// R06 팁 교환 완료 AUX
NOT
OR LOAD
OUT       M10036	// R06 원점 확인 요구
; L68
LOAD      M10031	// R01 원점 확인 요구
AND NOT   M10001	// R01 원점 확인 완료
OUT       M10138	// R01 (IN41) 원점확인

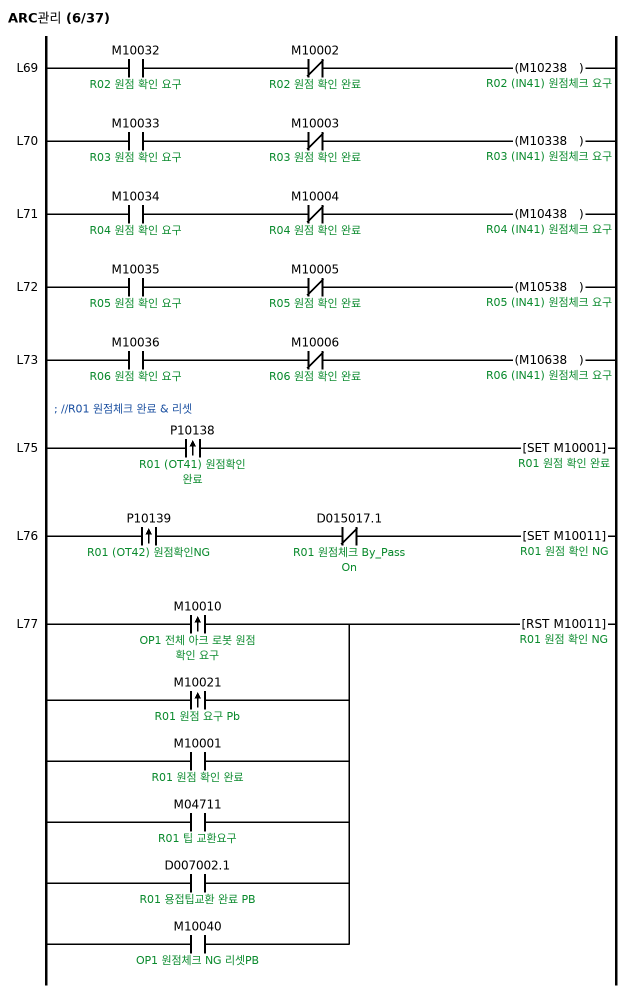
; L69
LOAD      M10032	// R02 원점 확인 요구
AND NOT   M10002	// R02 원점 확인 완료
OUT       M10238	// R02 (IN41) 원점체크 요구
; L70
LOAD      M10033	// R03 원점 확인 요구
AND NOT   M10003	// R03 원점 확인 완료
OUT       M10338	// R03 (IN41) 원점체크 요구
; L71
LOAD      M10034	// R04 원점 확인 요구
AND NOT   M10004	// R04 원점 확인 완료
OUT       M10438	// R04 (IN41) 원점체크 요구
; L72
LOAD      M10035	// R05 원점 확인 요구
AND NOT   M10005	// R05 원점 확인 완료
OUT       M10538	// R05 (IN41) 원점체크 요구
; L73
LOAD      M10036	// R06 원점 확인 요구
AND NOT   M10006	// R06 원점 확인 완료
OUT       M10638	// R06 (IN41) 원점체크 요구
//   //R01 원점체크 완료 & 리셋
; L75
LOADP     P10138	// R01 (OT41) 원점확인 완료
SET       M10001	// R01 원점 확인 완료
; L76
LOADP     P10139	// R01 (OT42) 원점확인NG
AND NOT   D015017.1	// R01 원점체크 By_Pass On
SET       M10011	// R01 원점 확인 NG
; L77
LOADP     M10010	// OP1 전체 아크 로봇 원점 확인 요구
ORP       M10021	// R01 원점 요구 Pb
OR        M10001	// R01 원점 확인 완료
OR        M04711	// R01 팁 교환요구
OR        D007002.1	// R01 용접팁교환 완료 PB
OR        M10040	// OP1 원점체크 NG 리셋PB
RST       M10011	// R01 원점 확인 NG

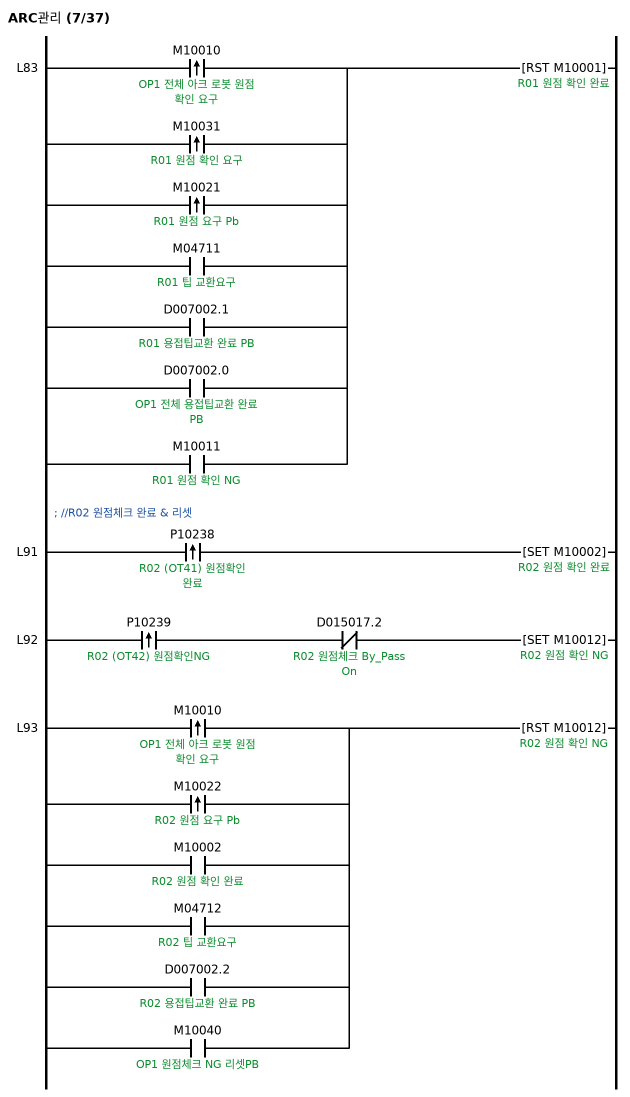
; L83
LOADP     M10010	// OP1 전체 아크 로봇 원점 확인 요구
ORP       M10031	// R01 원점 확인 요구
ORP       M10021	// R01 원점 요구 Pb
OR        M04711	// R01 팁 교환요구
OR        D007002.1	// R01 용접팁교환 완료 PB
OR        D007002.0	// OP1 전체 용접팁교환 완료 PB
OR        M10011	// R01 원점 확인 NG
RST       M10001	// R01 원점 확인 완료
//   //R02 원점체크 완료 & 리셋
; L91
LOADP     P10238	// R02 (OT41) 원점확인 완료
SET       M10002	// R02 원점 확인 완료
; L92
LOADP     P10239	// R02 (OT42) 원점확인NG
AND NOT   D015017.2	// R02 원점체크 By_Pass On
SET       M10012	// R02 원점 확인 NG
; L93
LOADP     M10010	// OP1 전체 아크 로봇 원점 확인 요구
ORP       M10022	// R02 원점 요구 Pb
OR        M10002	// R02 원점 확인 완료
OR        M04712	// R02 팁 교환요구
OR        D007002.2	// R02 용접팁교환 완료 PB
OR        M10040	// OP1 원점체크 NG 리셋PB
RST       M10012	// R02 원점 확인 NG

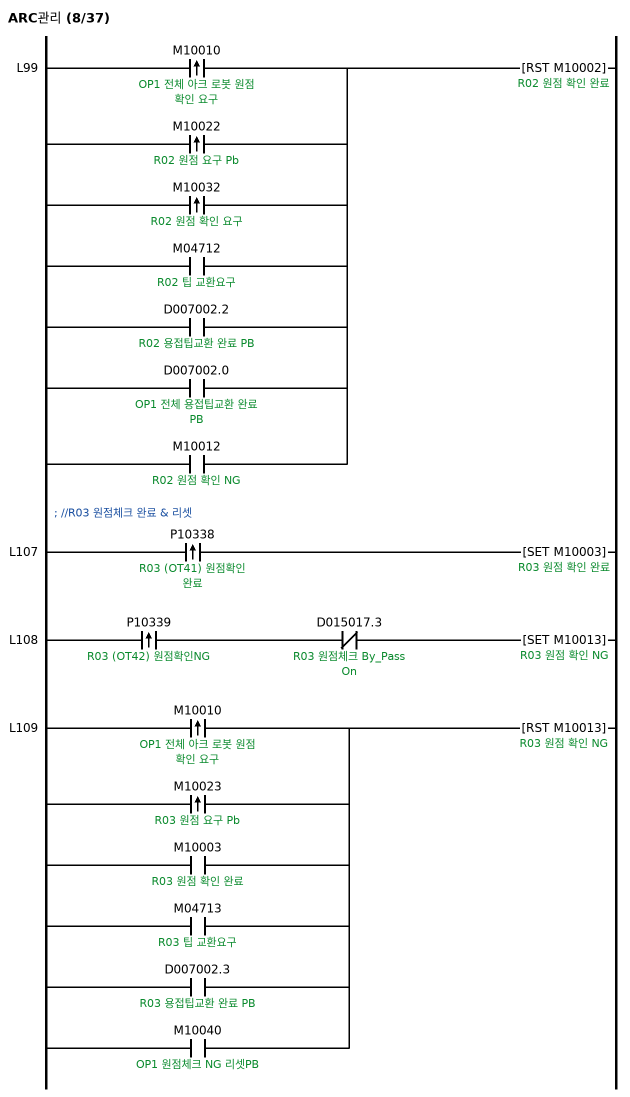
; L99
LOADP     M10010	// OP1 전체 아크 로봇 원점 확인 요구
ORP       M10022	// R02 원점 요구 Pb
ORP       M10032	// R02 원점 확인 요구
OR        M04712	// R02 팁 교환요구
OR        D007002.2	// R02 용접팁교환 완료 PB
OR        D007002.0	// OP1 전체 용접팁교환 완료 PB
OR        M10012	// R02 원점 확인 NG
RST       M10002	// R02 원점 확인 완료
//   //R03 원점체크 완료 & 리셋
; L107
LOADP     P10338	// R03 (OT41) 원점확인 완료
SET       M10003	// R03 원점 확인 완료
; L108
LOADP     P10339	// R03 (OT42) 원점확인NG
AND NOT   D015017.3	// R03 원점체크 By_Pass On
SET       M10013	// R03 원점 확인 NG
; L109
LOADP     M10010	// OP1 전체 아크 로봇 원점 확인 요구
ORP       M10023	// R03 원점 요구 Pb
OR        M10003	// R03 원점 확인 완료
OR        M04713	// R03 팁 교환요구
OR        D007002.3	// R03 용접팁교환 완료 PB
OR        M10040	// OP1 원점체크 NG 리셋PB
RST       M10013	// R03 원점 확인 NG

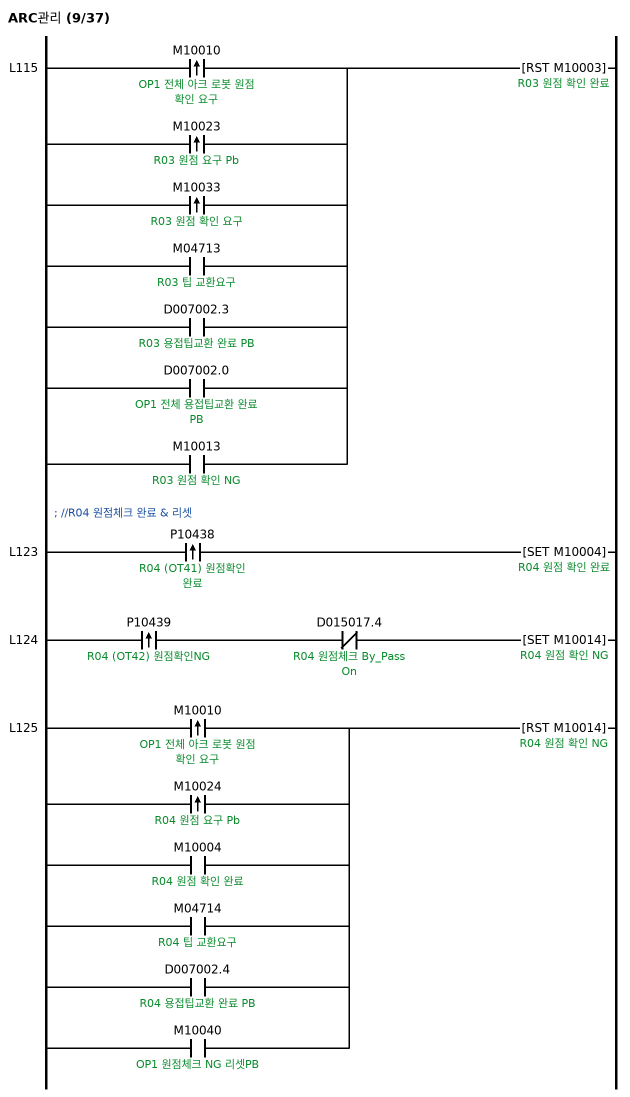
; L115
LOADP     M10010	// OP1 전체 아크 로봇 원점 확인 요구
ORP       M10023	// R03 원점 요구 Pb
ORP       M10033	// R03 원점 확인 요구
OR        M04713	// R03 팁 교환요구
OR        D007002.3	// R03 용접팁교환 완료 PB
OR        D007002.0	// OP1 전체 용접팁교환 완료 PB
OR        M10013	// R03 원점 확인 NG
RST       M10003	// R03 원점 확인 완료
//   //R04 원점체크 완료 & 리셋
; L123
LOADP     P10438	// R04 (OT41) 원점확인 완료
SET       M10004	// R04 원점 확인 완료
; L124
LOADP     P10439	// R04 (OT42) 원점확인NG
AND NOT   D015017.4	// R04 원점체크 By_Pass On
SET       M10014	// R04 원점 확인 NG
; L125
LOADP     M10010	// OP1 전체 아크 로봇 원점 확인 요구
ORP       M10024	// R04 원점 요구 Pb
OR        M10004	// R04 원점 확인 완료
OR        M04714	// R04 팁 교환요구
OR        D007002.4	// R04 용접팁교환 완료 PB
OR        M10040	// OP1 원점체크 NG 리셋PB
RST       M10014	// R04 원점 확인 NG

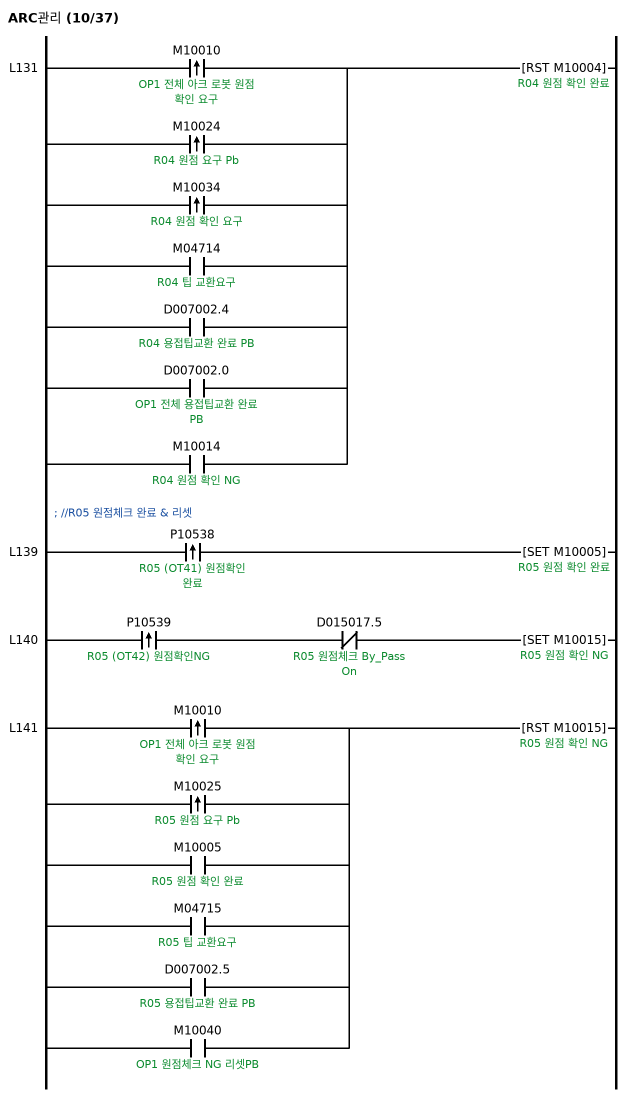
; L131
LOADP     M10010	// OP1 전체 아크 로봇 원점 확인 요구
ORP       M10024	// R04 원점 요구 Pb
ORP       M10034	// R04 원점 확인 요구
OR        M04714	// R04 팁 교환요구
OR        D007002.4	// R04 용접팁교환 완료 PB
OR        D007002.0	// OP1 전체 용접팁교환 완료 PB
OR        M10014	// R04 원점 확인 NG
RST       M10004	// R04 원점 확인 완료
//   //R05 원점체크 완료 & 리셋
; L139
LOADP     P10538	// R05 (OT41) 원점확인 완료
SET       M10005	// R05 원점 확인 완료
; L140
LOADP     P10539	// R05 (OT42) 원점확인NG
AND NOT   D015017.5	// R05 원점체크 By_Pass On
SET       M10015	// R05 원점 확인 NG
; L141
LOADP     M10010	// OP1 전체 아크 로봇 원점 확인 요구
ORP       M10025	// R05 원점 요구 Pb
OR        M10005	// R05 원점 확인 완료
OR        M04715	// R05 팁 교환요구
OR        D007002.5	// R05 용접팁교환 완료 PB
OR        M10040	// OP1 원점체크 NG 리셋PB
RST       M10015	// R05 원점 확인 NG

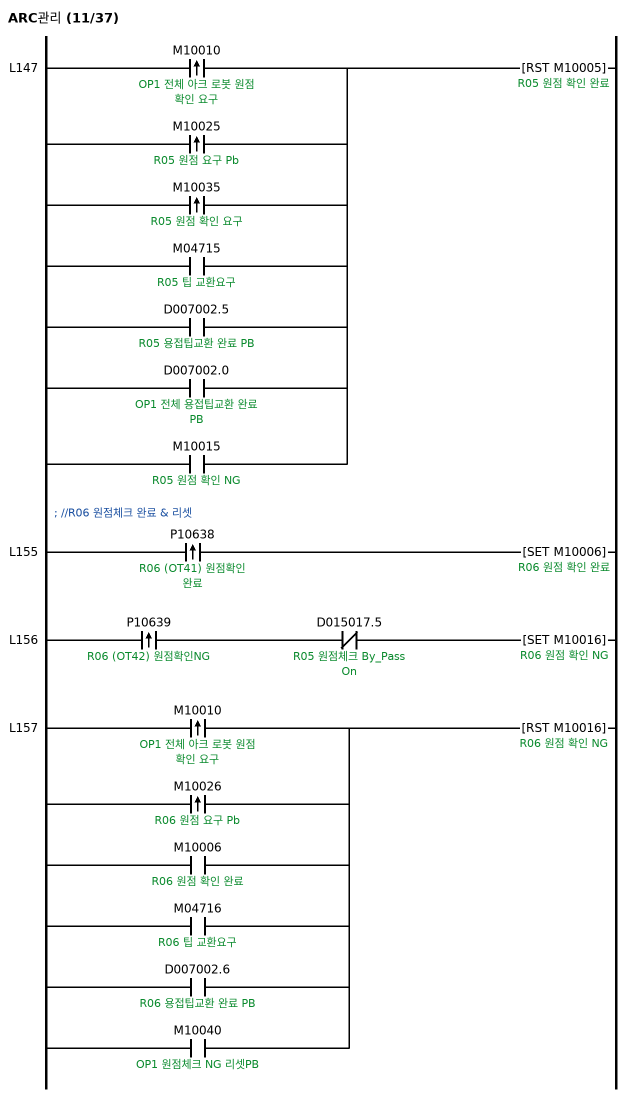
; L147
LOADP     M10010	// OP1 전체 아크 로봇 원점 확인 요구
ORP       M10025	// R05 원점 요구 Pb
ORP       M10035	// R05 원점 확인 요구
OR        M04715	// R05 팁 교환요구
OR        D007002.5	// R05 용접팁교환 완료 PB
OR        D007002.0	// OP1 전체 용접팁교환 완료 PB
OR        M10015	// R05 원점 확인 NG
RST       M10005	// R05 원점 확인 완료
//   //R06 원점체크 완료 & 리셋
; L155
LOADP     P10638	// R06 (OT41) 원점확인 완료
SET       M10006	// R06 원점 확인 완료
; L156
LOADP     P10639	// R06 (OT42) 원점확인NG
AND NOT   D015017.5	// R05 원점체크 By_Pass On
SET       M10016	// R06 원점 확인 NG
; L157
LOADP     M10010	// OP1 전체 아크 로봇 원점 확인 요구
ORP       M10026	// R06 원점 요구 Pb
OR        M10006	// R06 원점 확인 완료
OR        M04716	// R06 팁 교환요구
OR        D007002.6	// R06 용접팁교환 완료 PB
OR        M10040	// OP1 원점체크 NG 리셋PB
RST       M10016	// R06 원점 확인 NG

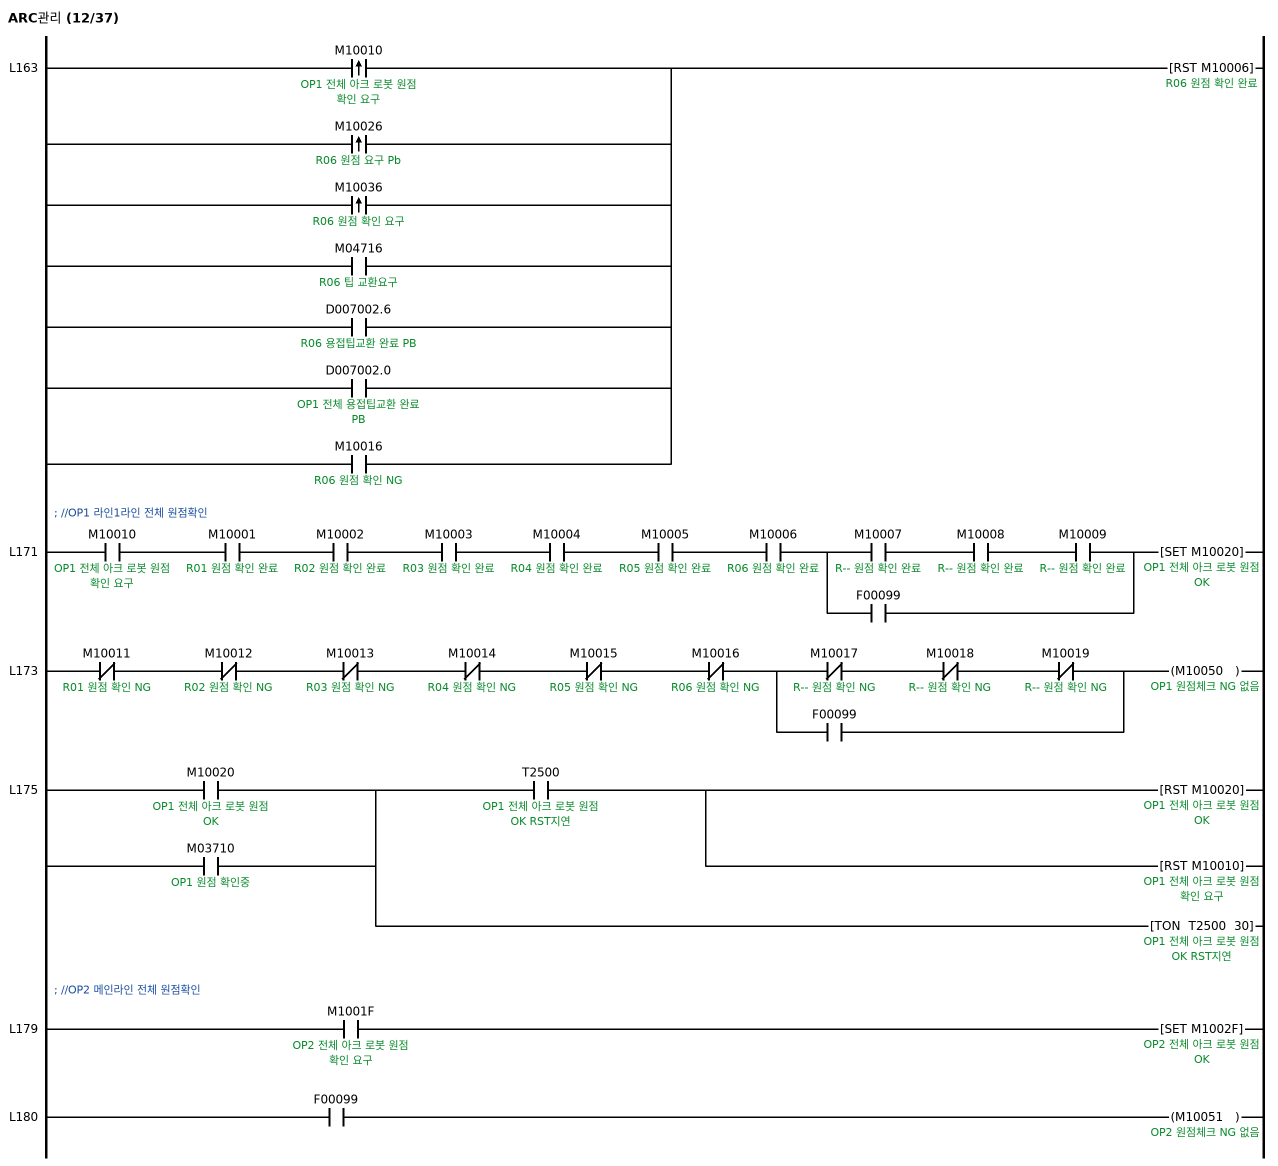
; L163
LOADP     M10010	// OP1 전체 아크 로봇 원점 확인 요구
ORP       M10026	// R06 원점 요구 Pb
ORP       M10036	// R06 원점 확인 요구
OR        M04716	// R06 팁 교환요구
OR        D007002.6	// R06 용접팁교환 완료 PB
OR        D007002.0	// OP1 전체 용접팁교환 완료 PB
OR        M10016	// R06 원점 확인 NG
RST       M10006	// R06 원점 확인 완료
//   //OP1 라인1라인 전체 원점확인
; L171
LOAD      M10010	// OP1 전체 아크 로봇 원점 확인 요구
AND       M10001	// R01 원점 확인 완료
AND       M10002	// R02 원점 확인 완료
AND       M10003	// R03 원점 확인 완료
AND       M10004	// R04 원점 확인 완료
AND       M10005	// R05 원점 확인 완료
AND       M10006	// R06 원점 확인 완료
LOAD      M10007	// R-- 원점 확인 완료
AND       M10008	// R-- 원점 확인 완료
AND       M10009	// R-- 원점 확인 완료
OR        F00099
AND LOAD
SET       M10020	// OP1 전체 아크 로봇 원점 OK
; L173
LOAD NOT  M10011	// R01 원점 확인 NG
AND NOT   M10012	// R02 원점 확인 NG
AND NOT   M10013	// R03 원점 확인 NG
AND NOT   M10014	// R04 원점 확인 NG
AND NOT   M10015	// R05 원점 확인 NG
AND NOT   M10016	// R06 원점 확인 NG
LOAD NOT  M10017	// R-- 원점 확인 NG
AND NOT   M10018	// R-- 원점 확인 NG
AND NOT   M10019	// R-- 원점 확인 NG
OR        F00099
AND LOAD
OUT       M10050	// OP1 원점체크 NG 없음
; L175
LOAD      M10020	// OP1 전체 아크 로봇 원점 OK
OR        M03710	// OP1 원점 확인중
MPUSH
AND       T2500	// OP1 전체 아크 로봇 원점 OK RST지연
RST       M10020	// OP1 전체 아크 로봇 원점 OK
RST       M10010	// OP1 전체 아크 로봇 원점 확인 요구
MPOP
TON       T2500 30	// OP1 전체 아크 로봇 원점 OK RST지연
//   //OP2 메인라인 전체 원점확인
; L179
LOAD      M1001F	// OP2 전체 아크 로봇 원점 확인 요구
SET       M1002F	// OP2 전체 아크 로봇 원점 OK
; L180
LOAD      F00099
OUT       M10051	// OP2 원점체크 NG 없음

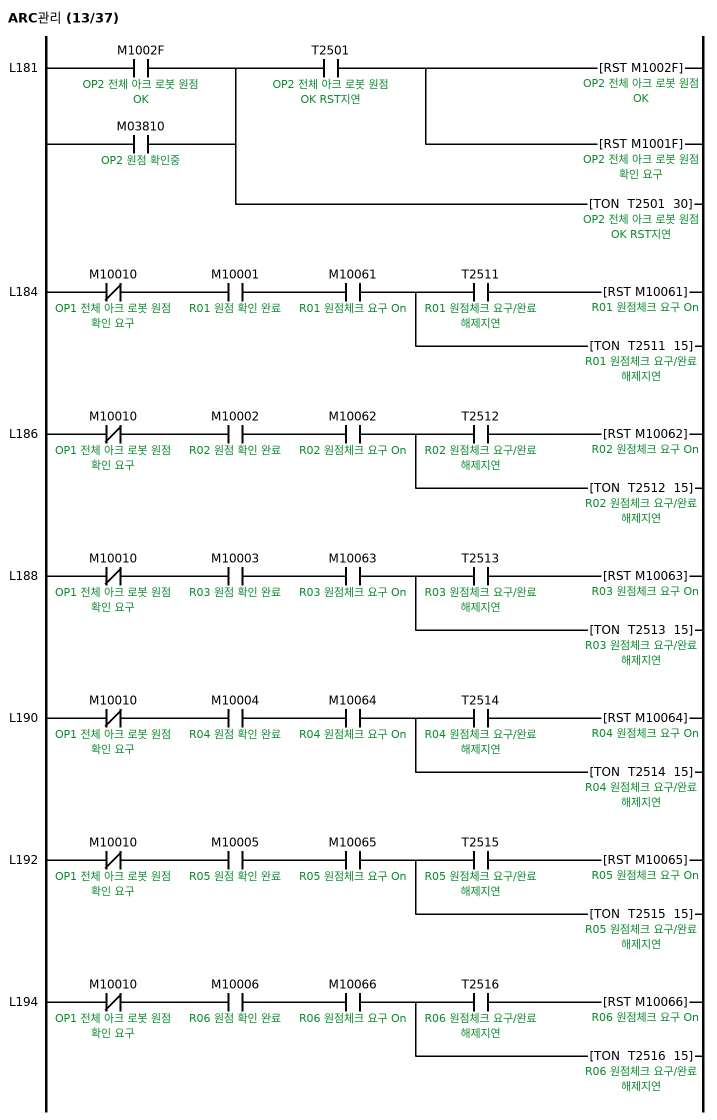
; L181
LOAD      M1002F	// OP2 전체 아크 로봇 원점 OK
OR        M03810	// OP2 원점 확인중
MPUSH
AND       T2501	// OP2 전체 아크 로봇 원점 OK RST지연
RST       M1002F	// OP2 전체 아크 로봇 원점 OK
RST       M1001F	// OP2 전체 아크 로봇 원점 확인 요구
MPOP
TON       T2501 30	// OP2 전체 아크 로봇 원점 OK RST지연
; L184
LOAD NOT  M10010	// OP1 전체 아크 로봇 원점 확인 요구
AND       M10001	// R01 원점 확인 완료
AND       M10061	// R01 원점체크 요구 On
MPUSH
AND       T2511	// R01 원점체크 요구/완료 해제지연
RST       M10061	// R01 원점체크 요구 On
MPOP
TON       T2511 15	// R01 원점체크 요구/완료 해제지연
; L186
LOAD NOT  M10010	// OP1 전체 아크 로봇 원점 확인 요구
AND       M10002	// R02 원점 확인 완료
AND       M10062	// R02 원점체크 요구 On
MPUSH
AND       T2512	// R02 원점체크 요구/완료 해제지연
RST       M10062	// R02 원점체크 요구 On
MPOP
TON       T2512 15	// R02 원점체크 요구/완료 해제지연
; L188
LOAD NOT  M10010	// OP1 전체 아크 로봇 원점 확인 요구
AND       M10003	// R03 원점 확인 완료
AND       M10063	// R03 원점체크 요구 On
MPUSH
AND       T2513	// R03 원점체크 요구/완료 해제지연
RST       M10063	// R03 원점체크 요구 On
MPOP
TON       T2513 15	// R03 원점체크 요구/완료 해제지연
; L190
LOAD NOT  M10010	// OP1 전체 아크 로봇 원점 확인 요구
AND       M10004	// R04 원점 확인 완료
AND       M10064	// R04 원점체크 요구 On
MPUSH
AND       T2514	// R04 원점체크 요구/완료 해제지연
RST       M10064	// R04 원점체크 요구 On
MPOP
TON       T2514 15	// R04 원점체크 요구/완료 해제지연
; L192
LOAD NOT  M10010	// OP1 전체 아크 로봇 원점 확인 요구
AND       M10005	// R05 원점 확인 완료
AND       M10065	// R05 원점체크 요구 On
MPUSH
AND       T2515	// R05 원점체크 요구/완료 해제지연
RST       M10065	// R05 원점체크 요구 On
MPOP
TON       T2515 15	// R05 원점체크 요구/완료 해제지연
; L194
LOAD NOT  M10010	// OP1 전체 아크 로봇 원점 확인 요구
AND       M10006	// R06 원점 확인 완료
AND       M10066	// R06 원점체크 요구 On
MPUSH
AND       T2516	// R06 원점체크 요구/완료 해제지연
RST       M10066	// R06 원점체크 요구 On
MPOP
TON       T2516 15	// R06 원점체크 요구/완료 해제지연

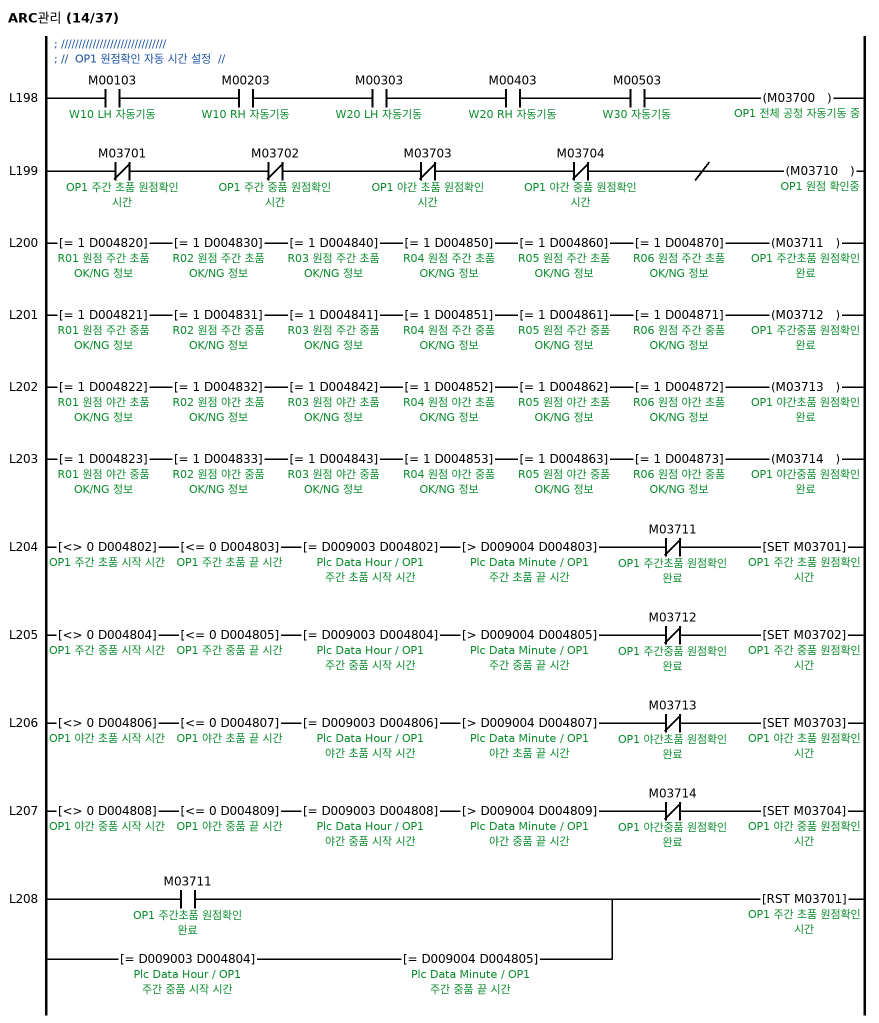
// //////////////////////////////
//   //  OP1 원점확인 자동 시간 설정  //
; L198
LOAD      M00103	// W10 LH 자동기동
AND       M00203	// W10 RH 자동기동
AND       M00303	// W20 LH 자동기동
AND       M00403	// W20 RH 자동기동
AND       M00503	// W30 자동기동
OUT       M03700	// OP1 전체 공정 자동기동 중
; L199
LOAD NOT  M03701	// OP1 주간 초품 원점확인 시간
AND NOT   M03702	// OP1 주간 중품 원점확인 시간
AND NOT   M03703	// OP1 야간 초품 원점확인 시간
AND NOT   M03704	// OP1 야간 중품 원점확인 시간
NOT
OUT       M03710	// OP1 원점 확인중
; L200
LOAD=     1 D004820	// R01 원점 주간 초품 OK/NG 정보
AND=      1 D004830	// R02 원점 주간 초품 OK/NG 정보
AND=      1 D004840	// R03 원점 주간 초품 OK/NG 정보
AND=      1 D004850	// R04 원점 주간 초품 OK/NG 정보
AND=      1 D004860	// R05 원점 주간 초품 OK/NG 정보
AND=      1 D004870	// R06 원점 주간 초품 OK/NG 정보
OUT       M03711	// OP1 주간초품 원점확인 완료
; L201
LOAD=     1 D004821	// R01 원점 주간 중품 OK/NG 정보
AND=      1 D004831	// R02 원점 주간 중품 OK/NG 정보
AND=      1 D004841	// R03 원점 주간 중품 OK/NG 정보
AND=      1 D004851	// R04 원점 주간 중품 OK/NG 정보
AND=      1 D004861	// R05 원점 주간 중품 OK/NG 정보
AND=      1 D004871	// R06 원점 주간 중품 OK/NG 정보
OUT       M03712	// OP1 주간중품 원점확인 완료
; L202
LOAD=     1 D004822	// R01 원점 야간 초품 OK/NG 정보
AND=      1 D004832	// R02 원점 야간 초품 OK/NG 정보
AND=      1 D004842	// R03 원점 야간 초품 OK/NG 정보
AND=      1 D004852	// R04 원점 야간 초품 OK/NG 정보
AND=      1 D004862	// R05 원점 야간 초품 OK/NG 정보
AND=      1 D004872	// R06 원점 야간 초품 OK/NG 정보
OUT       M03713	// OP1 야간초품 원점확인 완료
; L203
LOAD=     1 D004823	// R01 원점 야간 중품 OK/NG 정보
AND=      1 D004833	// R02 원점 야간 중품 OK/NG 정보
AND=      1 D004843	// R03 원점 야간 중품 OK/NG 정보
AND=      1 D004853	// R04 원점 야간 중품 OK/NG 정보
AND=      1 D004863	// R05 원점 야간 중품 OK/NG 정보
AND=      1 D004873	// R06 원점 야간 중품 OK/NG 정보
OUT       M03714	// OP1 야간중품 원점확인 완료
; L204
LOAD<>    0 D004802	// OP1 주간 초품 시작 시간
AND<=     0 D004803	// OP1 주간 초품 끝 시간
AND=      D009003 D004802	// Plc Data Hour / OP1 주간 초품 시작 시간
AND>      D009004 D004803	// Plc Data Minute / OP1 주간 초품 끝 시간
AND NOT   M03711	// OP1 주간초품 원점확인 완료
SET       M03701	// OP1 주간 초품 원점확인 시간
; L205
LOAD<>    0 D004804	// OP1 주간 중품 시작 시간
AND<=     0 D004805	// OP1 주간 중품 끝 시간
AND=      D009003 D004804	// Plc Data Hour / OP1 주간 중품 시작 시간
AND>      D009004 D004805	// Plc Data Minute / OP1 주간 중품 끝 시간
AND NOT   M03712	// OP1 주간중품 원점확인 완료
SET       M03702	// OP1 주간 중품 원점확인 시간
; L206
LOAD<>    0 D004806	// OP1 야간 초품 시작 시간
AND<=     0 D004807	// OP1 야간 초품 끝 시간
AND=      D009003 D004806	// Plc Data Hour / OP1 야간 초품 시작 시간
AND>      D009004 D004807	// Plc Data Minute / OP1 야간 초품 끝 시간
AND NOT   M03713	// OP1 야간초품 원점확인 완료
SET       M03703	// OP1 야간 초품 원점확인 시간
; L207
LOAD<>    0 D004808	// OP1 야간 중품 시작 시간
AND<=     0 D004809	// OP1 야간 중품 끝 시간
AND=      D009003 D004808	// Plc Data Hour / OP1 야간 중품 시작 시간
AND>      D009004 D004809	// Plc Data Minute / OP1 야간 중품 끝 시간
AND NOT   M03714	// OP1 야간중품 원점확인 완료
SET       M03704	// OP1 야간 중품 원점확인 시간
; L208
LOAD      M03711	// OP1 주간초품 원점확인 완료
LOAD=     D009003 D004804	// Plc Data Hour / OP1 주간 중품 시작 시간
AND=      D009004 D004805	// Plc Data Minute / OP1 주간 중품 끝 시간
OR LOAD
RST       M03701	// OP1 주간 초품 원점확인 시간

